// Mitsubishi GX Developer project: 11-1201_球閥後半段組立機_20140305   PLC: FX3U

PROGRAM MAIN
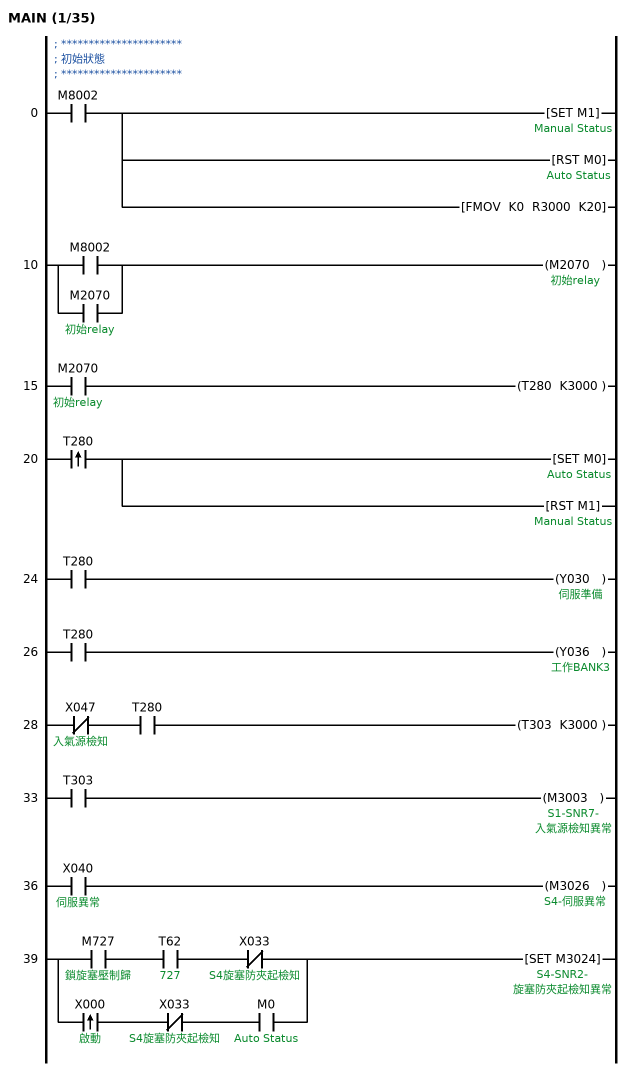
; **********************
; 初始狀態
; **********************
0     LD      M8002
      SET     M1  ; Manual Status
      RST     M0  ; Auto Status
      FMOV    K0 R3000 K20
10    LD      M8002
      OR      M2070  ; 初始relay
      OUT     M2070  ; 初始relay
15    LD      M2070  ; 初始relay
      OUT     T280 K3000
20    LDP     T280
      SET     M0  ; Auto Status
      RST     M1  ; Manual Status
24    LD      T280
      OUT     Y030  ; 伺服準備
26    LD      T280
      OUT     Y036  ; 工作BANK3
28    LDI     X047  ; 入氣源檢知
      AND     T280
      OUT     T303 K3000
33    LD      T303
      OUT     M3003  ; S1-SNR7-入氣源檢知異常
36    LD      X040  ; 伺服異常
      OUT     M3026  ; S4-伺服異常
39    LD      M727  ; 鎖旋塞壓制歸
      AND     T62  ; 727
      ANI     X033  ; S4旋塞防夾起檢知
      LDP     X000  ; 啟動
      ANI     X033  ; S4旋塞防夾起檢知
      AND     M0  ; Auto Status
      ORB
      SET     M3024  ; S4-SNR2-旋塞防夾起檢知異常
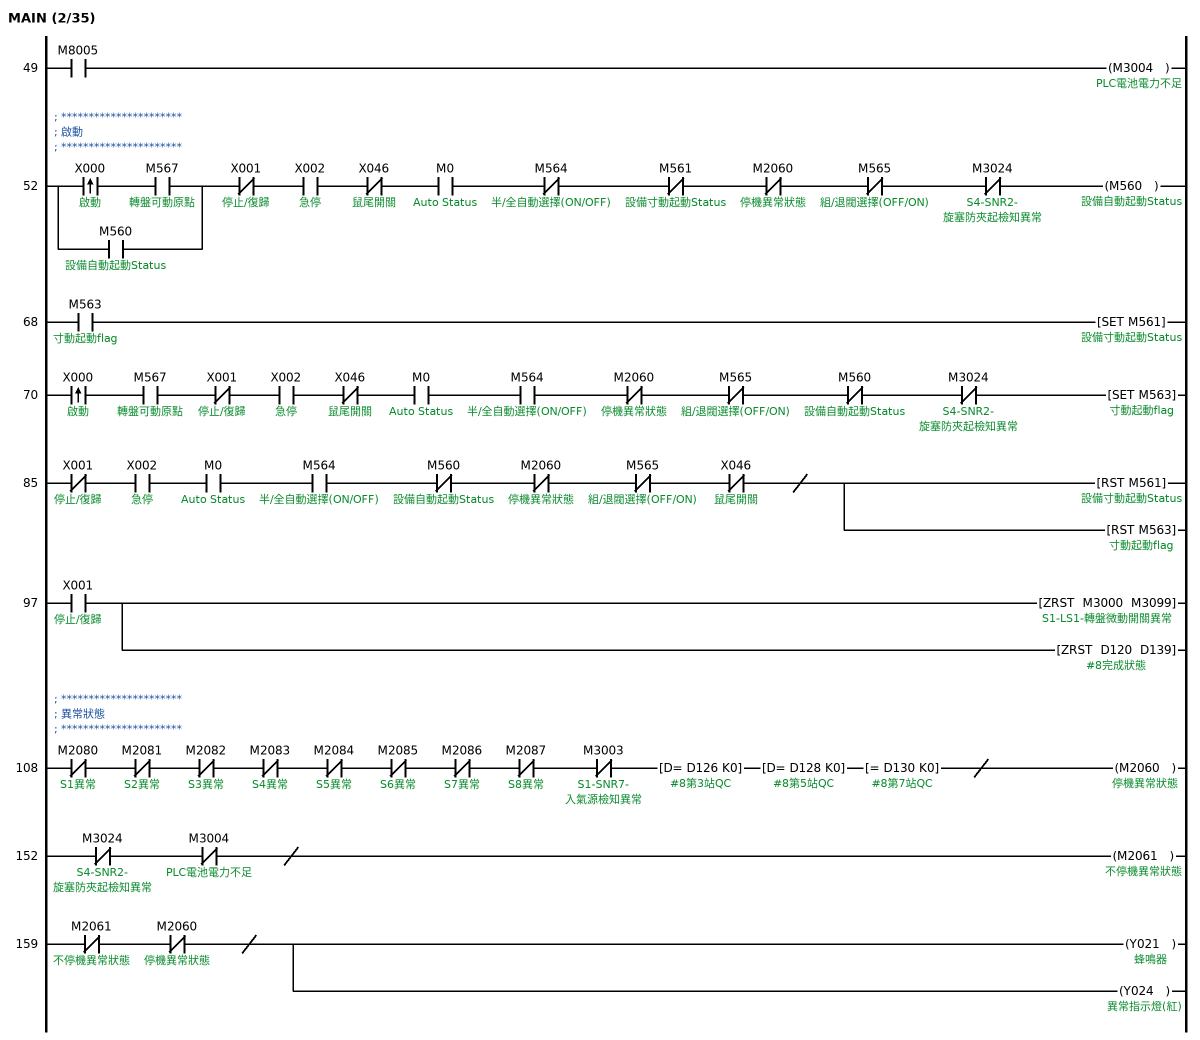
49    LD      M8005
      OUT     M3004  ; PLC電池電力不足
; **********************
; 啟動
; **********************
52    LDP     X000  ; 啟動
      AND     M567  ; 轉盤可動原點
      OR      M560  ; 設備自動起動Status
      ANI     X001  ; 停止/復歸
      AND     X002  ; 急停
      ANI     X046  ; 鼠尾開關
      AND     M0  ; Auto Status
      ANI     M564  ; 半/全自動選擇(ON/OFF)
      ANI     M561  ; 設備寸動起動Status
      ANI     M2060  ; 停機異常狀態
      ANI     M565  ; 組/退閥選擇(OFF/ON)
      ANI     M3024  ; S4-SNR2-旋塞防夾起檢知異常
      OUT     M560  ; 設備自動起動Status
68    LD      M563  ; 寸動起動flag
      SET     M561  ; 設備寸動起動Status
70    LDP     X000  ; 啟動
      AND     M567  ; 轉盤可動原點
      ANI     X001  ; 停止/復歸
      AND     X002  ; 急停
      ANI     X046  ; 鼠尾開關
      AND     M0  ; Auto Status
      AND     M564  ; 半/全自動選擇(ON/OFF)
      ANI     M2060  ; 停機異常狀態
      ANI     M565  ; 組/退閥選擇(OFF/ON)
      ANI     M560  ; 設備自動起動Status
      ANI     M3024  ; S4-SNR2-旋塞防夾起檢知異常
      SET     M563  ; 寸動起動flag
85    LDI     X001  ; 停止/復歸
      AND     X002  ; 急停
      AND     M0  ; Auto Status
      AND     M564  ; 半/全自動選擇(ON/OFF)
      ANI     M560  ; 設備自動起動Status
      ANI     M2060  ; 停機異常狀態
      ANI     M565  ; 組/退閥選擇(OFF/ON)
      ANI     X046  ; 鼠尾開關
      INV
      RST     M561  ; 設備寸動起動Status
      RST     M563  ; 寸動起動flag
97    LD      X001  ; 停止/復歸
      ZRST    M3000 M3099  ; S1-LS1-轉盤微動開關異常
      ZRST    D120 D139  ; #8完成狀態
; **********************
; 異常狀態
; **********************
108   LDI     M2080  ; S1異常
      ANI     M2081  ; S2異常
      ANI     M2082  ; S3異常
      ANI     M2083  ; S4異常
      ANI     M2084  ; S5異常
      ANI     M2085  ; S6異常
      ANI     M2086  ; S7異常
      ANI     M2087  ; S8異常
      ANI     M3003  ; S1-SNR7-入氣源檢知異常
      ANDD=   D126 K0  ; #8第3站QC
      ANDD=   D128 K0  ; #8第5站QC
      AND=    D130 K0  ; #8第7站QC
      INV
      OUT     M2060  ; 停機異常狀態
152   LDI     M3024  ; S4-SNR2-旋塞防夾起檢知異常
      ANI     M3004  ; PLC電池電力不足
      INV
      OUT     M2061  ; 不停機異常狀態
159   LDI     M2061  ; 不停機異常狀態
      ANI     M2060  ; 停機異常狀態
      INV
      OUT     Y021  ; 蜂鳴器
      OUT     Y024  ; 異常指示燈(紅)
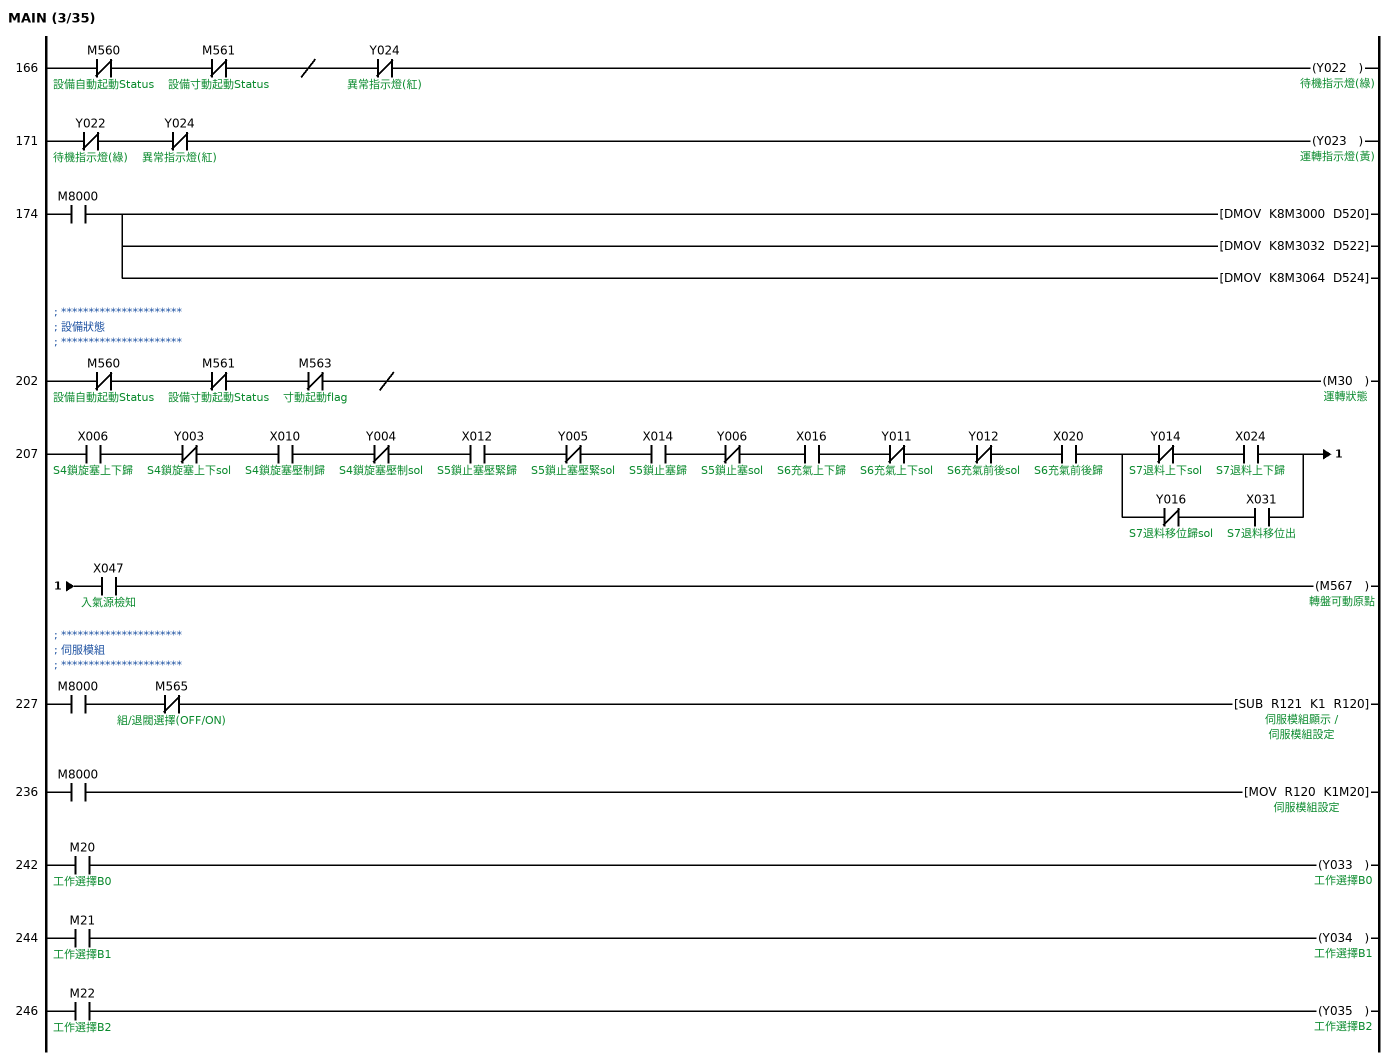
166   LDI     M560  ; 設備自動起動Status
      ANI     M561  ; 設備寸動起動Status
      INV
      ANI     Y024  ; 異常指示燈(紅)
      OUT     Y022  ; 待機指示燈(綠)
171   LDI     Y022  ; 待機指示燈(綠)
      ANI     Y024  ; 異常指示燈(紅)
      OUT     Y023  ; 運轉指示燈(黃)
174   LD      M8000
      DMOV    K8M3000 D520
      DMOV    K8M3032 D522
      DMOV    K8M3064 D524  ; S6-LS16-充氣旋轉歸異常
; **********************
; 設備狀態
; **********************
202   LDI     M560  ; 設備自動起動Status
      ANI     M561  ; 設備寸動起動Status
      ANI     M563  ; 寸動起動flag
      INV
      OUT     M30  ; 運轉狀態
207   LD      X006  ; S4鎖旋塞上下歸
      ANI     Y003  ; S4鎖旋塞上下sol
      AND     X010  ; S4鎖旋塞壓制歸
      ANI     Y004  ; S4鎖旋塞壓制sol
      AND     X012  ; S5鎖止塞壓緊歸
      ANI     Y005  ; S5鎖止塞壓緊sol
      AND     X014  ; S5鎖止塞歸
      ANI     Y006  ; S5鎖止塞sol
      AND     X016  ; S6充氣上下歸
      ANI     Y011  ; S6充氣上下sol
      ANI     Y012  ; S6充氣前後sol
      AND     X020  ; S6充氣前後歸
      LDI     Y014  ; S7退料上下sol
      AND     X024  ; S7退料上下歸
      LDI     Y016  ; S7退料移位歸sol
      AND     X031  ; S7退料移位出
      ORB
      ANB
      AND     X047  ; 入氣源檢知
      OUT     M567  ; 轉盤可動原點
; **********************
; 伺服模組
; **********************
227   LD      M8000
      ANI     M565  ; 組/退閥選擇(OFF/ON)
      SUB     R121 K1 R120  ; 伺服模組顯示 / 伺服模組設定
236   LD      M8000
      MOV     R120 K1M20  ; 工作選擇B0
242   LD      M20  ; 工作選擇B0
      OUT     Y033  ; 工作選擇B0
244   LD      M21  ; 工作選擇B1
      OUT     Y034  ; 工作選擇B1
246   LD      M22  ; 工作選擇B2
      OUT     Y035  ; 工作選擇B2
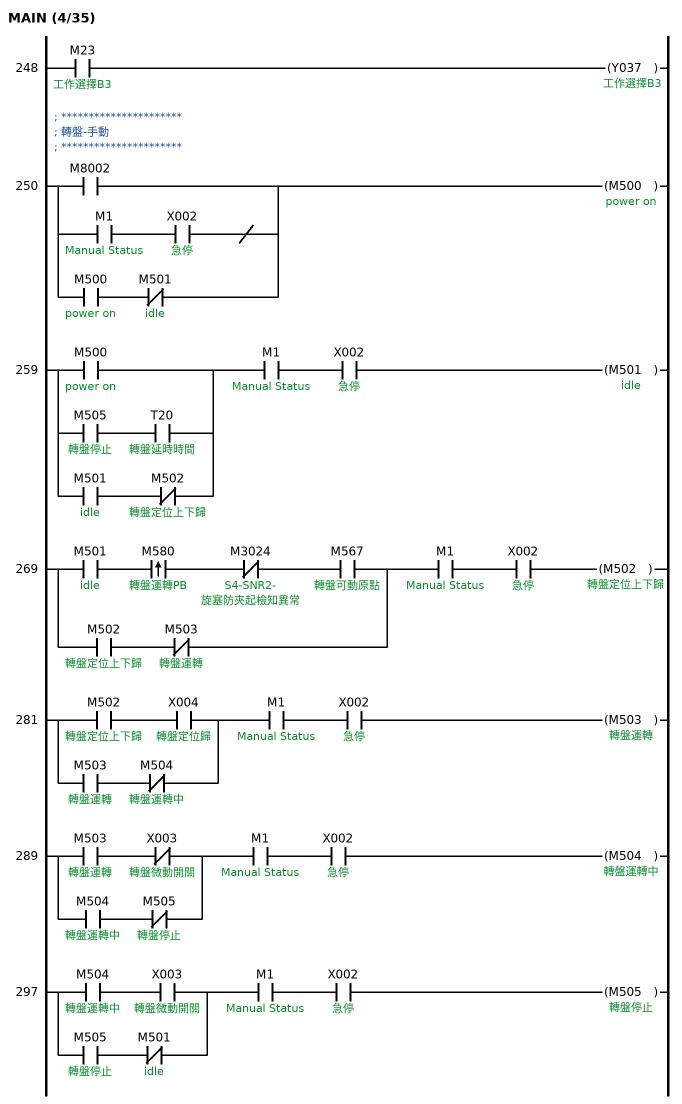
248   LD      M23  ; 工作選擇B3
      OUT     Y037  ; 工作選擇B3
; **********************
; 轉盤-手動
; **********************
250   LD      M8002
      LD      M1  ; Manual Status
      AND     X002  ; 急停
      INV
      ORB
      LD      M500  ; power on
      ANI     M501  ; idle
      ORB
      OUT     M500  ; power on
259   LD      M500  ; power on
      LD      M505  ; 轉盤停止
      AND     T20  ; 轉盤延時時間
      ORB
      LD      M501  ; idle
      ANI     M502  ; 轉盤定位上下歸
      ORB
      AND     M1  ; Manual Status
      AND     X002  ; 急停
      OUT     M501  ; idle
269   LD      M501  ; idle
      ANDP    M580  ; 轉盤運轉PB
      ANI     M3024  ; S4-SNR2-旋塞防夾起檢知異常
      AND     M567  ; 轉盤可動原點
      LD      M502  ; 轉盤定位上下歸
      ANI     M503  ; 轉盤運轉
      ORB
      AND     M1  ; Manual Status
      AND     X002  ; 急停
      OUT     M502  ; 轉盤定位上下歸
281   LD      M502  ; 轉盤定位上下歸
      AND     X004  ; 轉盤定位歸
      LD      M503  ; 轉盤運轉
      ANI     M504  ; 轉盤運轉中
      ORB
      AND     M1  ; Manual Status
      AND     X002  ; 急停
      OUT     M503  ; 轉盤運轉
289   LD      M503  ; 轉盤運轉
      ANI     X003  ; 轉盤微動開關
      LD      M504  ; 轉盤運轉中
      ANI     M505  ; 轉盤停止
      ORB
      AND     M1  ; Manual Status
      AND     X002  ; 急停
      OUT     M504  ; 轉盤運轉中
297   LD      M504  ; 轉盤運轉中
      AND     X003  ; 轉盤微動開關
      LD      M505  ; 轉盤停止
      ANI     M501  ; idle
      ORB
      AND     M1  ; Manual Status
      AND     X002  ; 急停
      OUT     M505  ; 轉盤停止
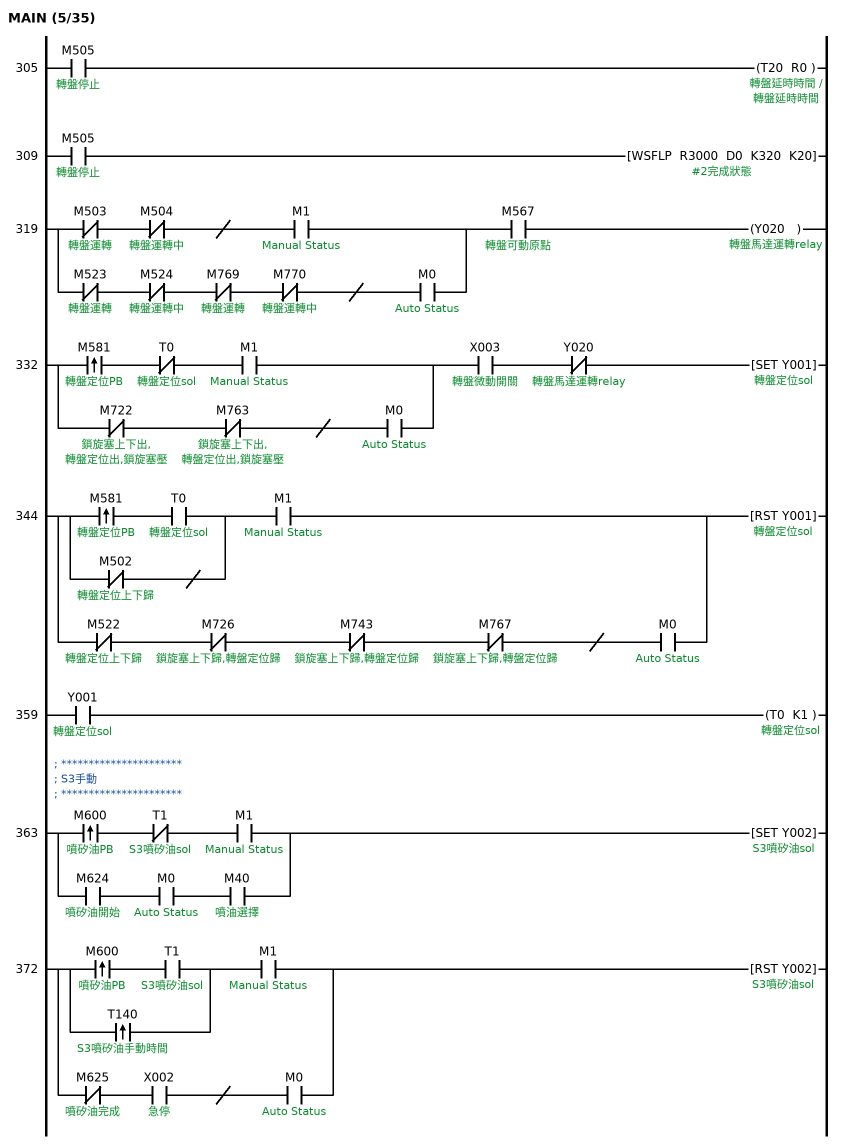
305   LD      M505  ; 轉盤停止
      OUT     T20 R0  ; 轉盤延時時間 / 轉盤延時時間
309   LD      M505  ; 轉盤停止
      WSFLP   R3000 D0 K320 K20  ; #2完成狀態
319   LDI     M503  ; 轉盤運轉
      ANI     M504  ; 轉盤運轉中
      INV
      AND     M1  ; Manual Status
      LDI     M523  ; 轉盤運轉
      ANI     M524  ; 轉盤運轉中
      ANI     M769  ; 轉盤運轉
      ANI     M770  ; 轉盤運轉中
      INV
      AND     M0  ; Auto Status
      ORB
      AND     M567  ; 轉盤可動原點
      OUT     Y020  ; 轉盤馬達運轉relay
332   LDP     M581  ; 轉盤定位PB
      ANI     T0  ; 轉盤定位sol
      AND     M1  ; Manual Status
      LDI     M722  ; 鎖旋塞上下出,轉盤定位出,鎖旋塞壓
      ANI     M763  ; 鎖旋塞上下出,轉盤定位出,鎖旋塞壓
      INV
      AND     M0  ; Auto Status
      ORB
      AND     X003  ; 轉盤微動開關
      ANI     Y020  ; 轉盤馬達運轉relay
      SET     Y001  ; 轉盤定位sol
344   LDP     M581  ; 轉盤定位PB
      AND     T0  ; 轉盤定位sol
      LDI     M502  ; 轉盤定位上下歸
      INV
      ORB
      AND     M1  ; Manual Status
      LDI     M522  ; 轉盤定位上下歸
      ANI     M726  ; 鎖旋塞上下歸,轉盤定位歸
      ANI     M743  ; 鎖旋塞上下歸,轉盤定位歸
      ANI     M767  ; 鎖旋塞上下歸,轉盤定位歸
      INV
      AND     M0  ; Auto Status
      ORB
      RST     Y001  ; 轉盤定位sol
359   LD      Y001  ; 轉盤定位sol
      OUT     T0 K1  ; 轉盤定位sol
; **********************
; S3手動
; **********************
363   LDP     M600  ; 噴矽油PB
      ANI     T1  ; S3噴矽油sol
      AND     M1  ; Manual Status
      LD      M624  ; 噴矽油開始
      AND     M0  ; Auto Status
      AND     M40  ; 噴油選擇
      ORB
      SET     Y002  ; S3噴矽油sol
372   LDP     M600  ; 噴矽油PB
      AND     T1  ; S3噴矽油sol
      ORP     T140  ; S3噴矽油手動時間
      AND     M1  ; Manual Status
      LDI     M625  ; 噴矽油完成
      AND     X002  ; 急停
      INV
      AND     M0  ; Auto Status
      ORB
      RST     Y002  ; S3噴矽油sol
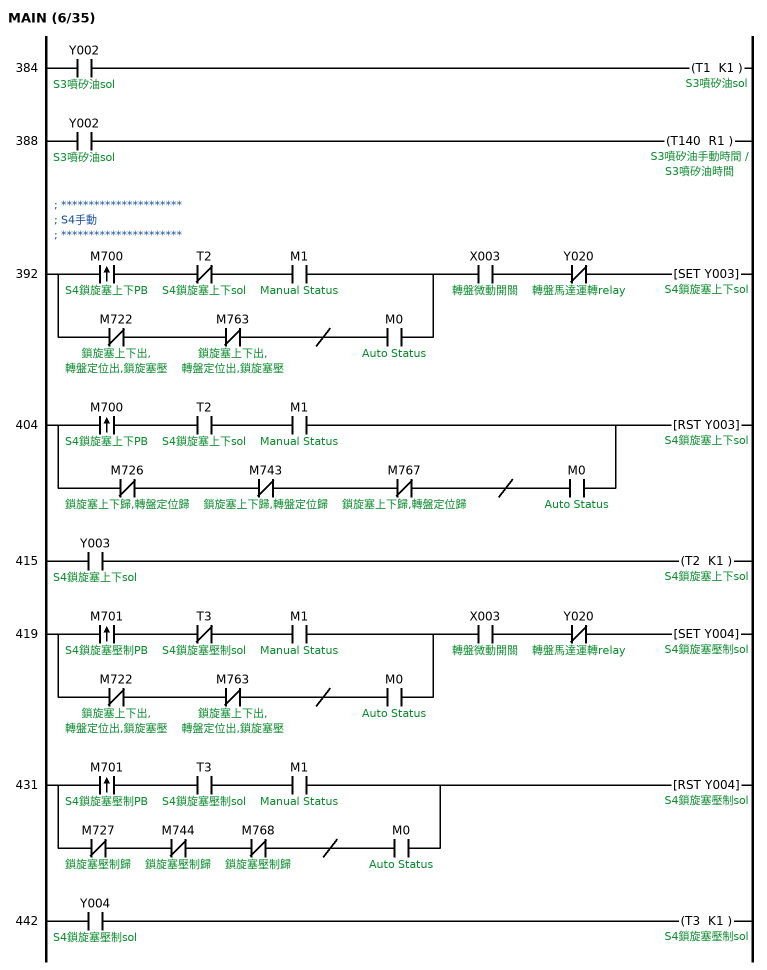
384   LD      Y002  ; S3噴矽油sol
      OUT     T1 K1  ; S3噴矽油sol
388   LD      Y002  ; S3噴矽油sol
      OUT     T140 R1  ; S3噴矽油手動時間 / S3噴矽油時間
; **********************
; S4手動
; **********************
392   LDP     M700  ; S4鎖旋塞上下PB
      ANI     T2  ; S4鎖旋塞上下sol
      AND     M1  ; Manual Status
      LDI     M722  ; 鎖旋塞上下出,轉盤定位出,鎖旋塞壓
      ANI     M763  ; 鎖旋塞上下出,轉盤定位出,鎖旋塞壓
      INV
      AND     M0  ; Auto Status
      ORB
      AND     X003  ; 轉盤微動開關
      ANI     Y020  ; 轉盤馬達運轉relay
      SET     Y003  ; S4鎖旋塞上下sol
404   LDP     M700  ; S4鎖旋塞上下PB
      AND     T2  ; S4鎖旋塞上下sol
      AND     M1  ; Manual Status
      LDI     M726  ; 鎖旋塞上下歸,轉盤定位歸
      ANI     M743  ; 鎖旋塞上下歸,轉盤定位歸
      ANI     M767  ; 鎖旋塞上下歸,轉盤定位歸
      INV
      AND     M0  ; Auto Status
      ORB
      RST     Y003  ; S4鎖旋塞上下sol
415   LD      Y003  ; S4鎖旋塞上下sol
      OUT     T2 K1  ; S4鎖旋塞上下sol
419   LDP     M701  ; S4鎖旋塞壓制PB
      ANI     T3  ; S4鎖旋塞壓制sol
      AND     M1  ; Manual Status
      LDI     M722  ; 鎖旋塞上下出,轉盤定位出,鎖旋塞壓
      ANI     M763  ; 鎖旋塞上下出,轉盤定位出,鎖旋塞壓
      INV
      AND     M0  ; Auto Status
      ORB
      AND     X003  ; 轉盤微動開關
      ANI     Y020  ; 轉盤馬達運轉relay
      SET     Y004  ; S4鎖旋塞壓制sol
431   LDP     M701  ; S4鎖旋塞壓制PB
      AND     T3  ; S4鎖旋塞壓制sol
      AND     M1  ; Manual Status
      LDI     M727  ; 鎖旋塞壓制歸
      ANI     M744  ; 鎖旋塞壓制歸
      ANI     M768  ; 鎖旋塞壓制歸
      INV
      AND     M0  ; Auto Status
      ORB
      RST     Y004  ; S4鎖旋塞壓制sol
442   LD      Y004  ; S4鎖旋塞壓制sol
      OUT     T3 K1  ; S4鎖旋塞壓制sol
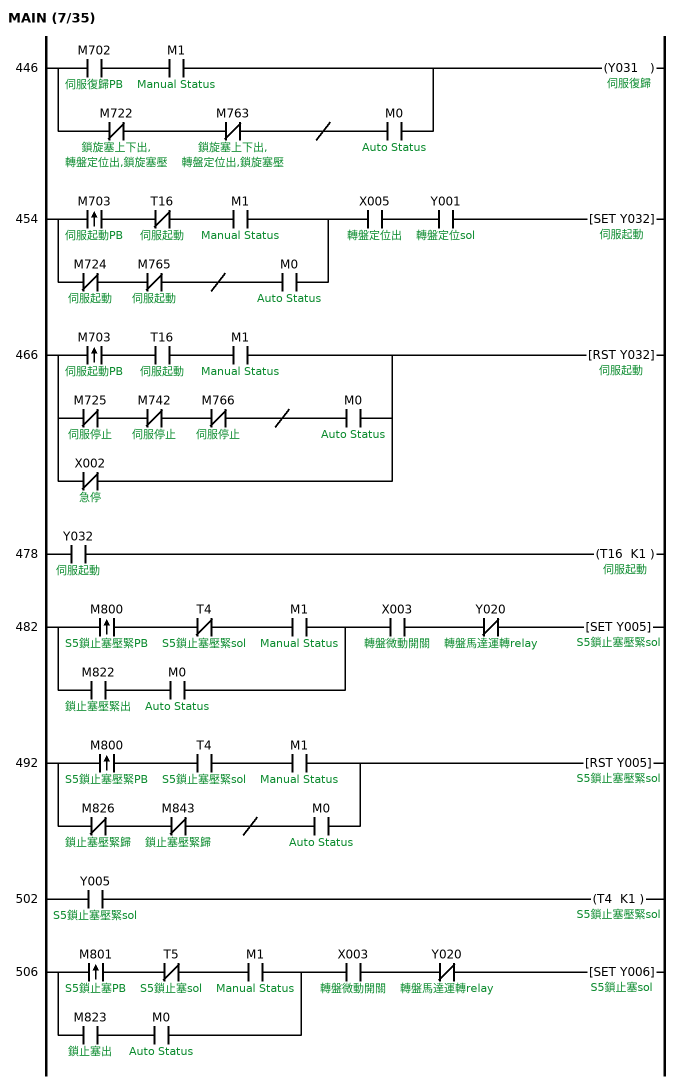
446   LD      M702  ; 伺服復歸PB
      AND     M1  ; Manual Status
      LDI     M722  ; 鎖旋塞上下出,轉盤定位出,鎖旋塞壓
      ANI     M763  ; 鎖旋塞上下出,轉盤定位出,鎖旋塞壓
      INV
      AND     M0  ; Auto Status
      ORB
      OUT     Y031  ; 伺服復歸
454   LDP     M703  ; 伺服起動PB
      ANI     T16  ; 伺服起動
      AND     M1  ; Manual Status
      LDI     M724  ; 伺服起動
      ANI     M765  ; 伺服起動
      INV
      AND     M0  ; Auto Status
      ORB
      AND     X005  ; 轉盤定位出
      AND     Y001  ; 轉盤定位sol
      SET     Y032  ; 伺服起動
466   LDP     M703  ; 伺服起動PB
      AND     T16  ; 伺服起動
      AND     M1  ; Manual Status
      LDI     M725  ; 伺服停止
      ANI     M742  ; 伺服停止
      ANI     M766  ; 伺服停止
      INV
      AND     M0  ; Auto Status
      ORB
      ORI     X002  ; 急停
      RST     Y032  ; 伺服起動
478   LD      Y032  ; 伺服起動
      OUT     T16 K1  ; 伺服起動
482   LDP     M800  ; S5鎖止塞壓緊PB
      ANI     T4  ; S5鎖止塞壓緊sol
      AND     M1  ; Manual Status
      LD      M822  ; 鎖止塞壓緊出
      AND     M0  ; Auto Status
      ORB
      AND     X003  ; 轉盤微動開關
      ANI     Y020  ; 轉盤馬達運轉relay
      SET     Y005  ; S5鎖止塞壓緊sol
492   LDP     M800  ; S5鎖止塞壓緊PB
      AND     T4  ; S5鎖止塞壓緊sol
      AND     M1  ; Manual Status
      LDI     M826  ; 鎖止塞壓緊歸
      ANI     M843  ; 鎖止塞壓緊歸
      INV
      AND     M0  ; Auto Status
      ORB
      RST     Y005  ; S5鎖止塞壓緊sol
502   LD      Y005  ; S5鎖止塞壓緊sol
      OUT     T4 K1  ; S5鎖止塞壓緊sol
506   LDP     M801  ; S5鎖止塞PB
      ANI     T5  ; S5鎖止塞sol
      AND     M1  ; Manual Status
      LD      M823  ; 鎖止塞出
      AND     M0  ; Auto Status
      ORB
      AND     X003  ; 轉盤微動開關
      ANI     Y020  ; 轉盤馬達運轉relay
      SET     Y006  ; S5鎖止塞sol
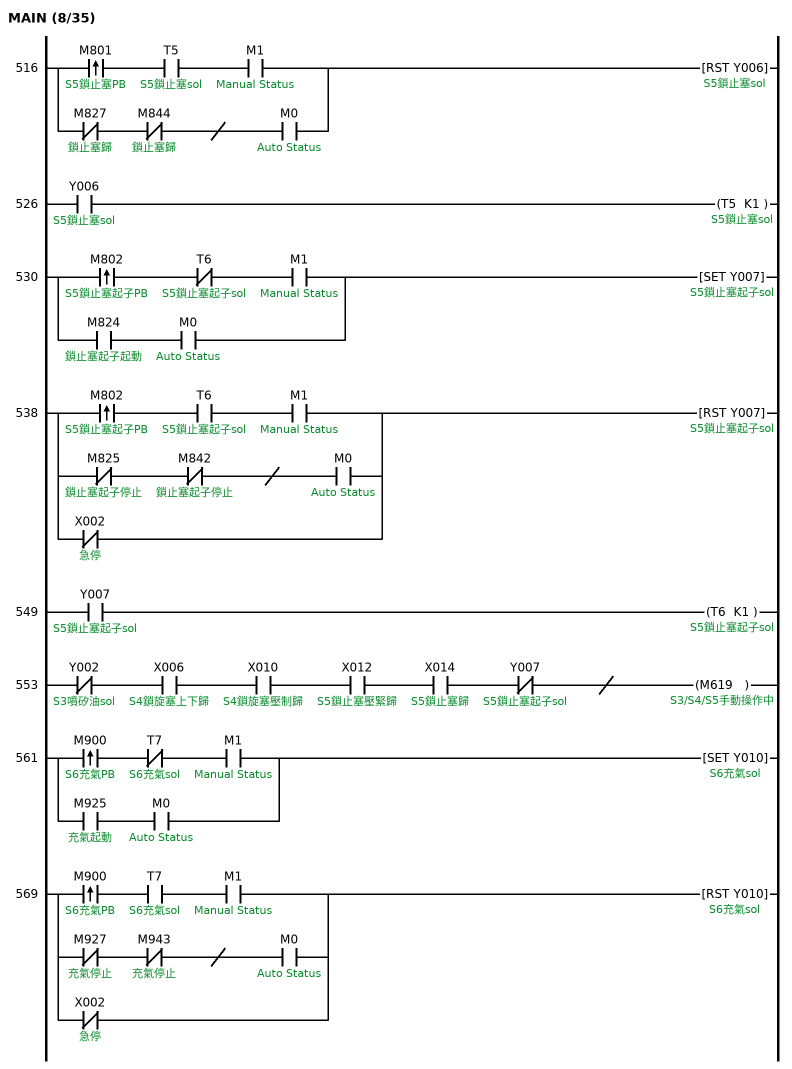
516   LDP     M801  ; S5鎖止塞PB
      AND     T5  ; S5鎖止塞sol
      AND     M1  ; Manual Status
      LDI     M827  ; 鎖止塞歸
      ANI     M844  ; 鎖止塞歸
      INV
      AND     M0  ; Auto Status
      ORB
      RST     Y006  ; S5鎖止塞sol
526   LD      Y006  ; S5鎖止塞sol
      OUT     T5 K1  ; S5鎖止塞sol
530   LDP     M802  ; S5鎖止塞起子PB
      ANI     T6  ; S5鎖止塞起子sol
      AND     M1  ; Manual Status
      LD      M824  ; 鎖止塞起子起動
      AND     M0  ; Auto Status
      ORB
      SET     Y007  ; S5鎖止塞起子sol
538   LDP     M802  ; S5鎖止塞起子PB
      AND     T6  ; S5鎖止塞起子sol
      AND     M1  ; Manual Status
      LDI     M825  ; 鎖止塞起子停止
      ANI     M842  ; 鎖止塞起子停止
      INV
      AND     M0  ; Auto Status
      ORB
      ORI     X002  ; 急停
      RST     Y007  ; S5鎖止塞起子sol
549   LD      Y007  ; S5鎖止塞起子sol
      OUT     T6 K1  ; S5鎖止塞起子sol
553   LDI     Y002  ; S3噴矽油sol
      AND     X006  ; S4鎖旋塞上下歸
      AND     X010  ; S4鎖旋塞壓制歸
      AND     X012  ; S5鎖止塞壓緊歸
      AND     X014  ; S5鎖止塞歸
      ANI     Y007  ; S5鎖止塞起子sol
      INV
      OUT     M619  ; S3/S4/S5手動操作中
561   LDP     M900  ; S6充氣PB
      ANI     T7  ; S6充氣sol
      AND     M1  ; Manual Status
      LD      M925  ; 充氣起動
      AND     M0  ; Auto Status
      ORB
      SET     Y010  ; S6充氣sol
569   LDP     M900  ; S6充氣PB
      AND     T7  ; S6充氣sol
      AND     M1  ; Manual Status
      LDI     M927  ; 充氣停止
      ANI     M943  ; 充氣停止
      INV
      AND     M0  ; Auto Status
      ORB
      ORI     X002  ; 急停
      RST     Y010  ; S6充氣sol
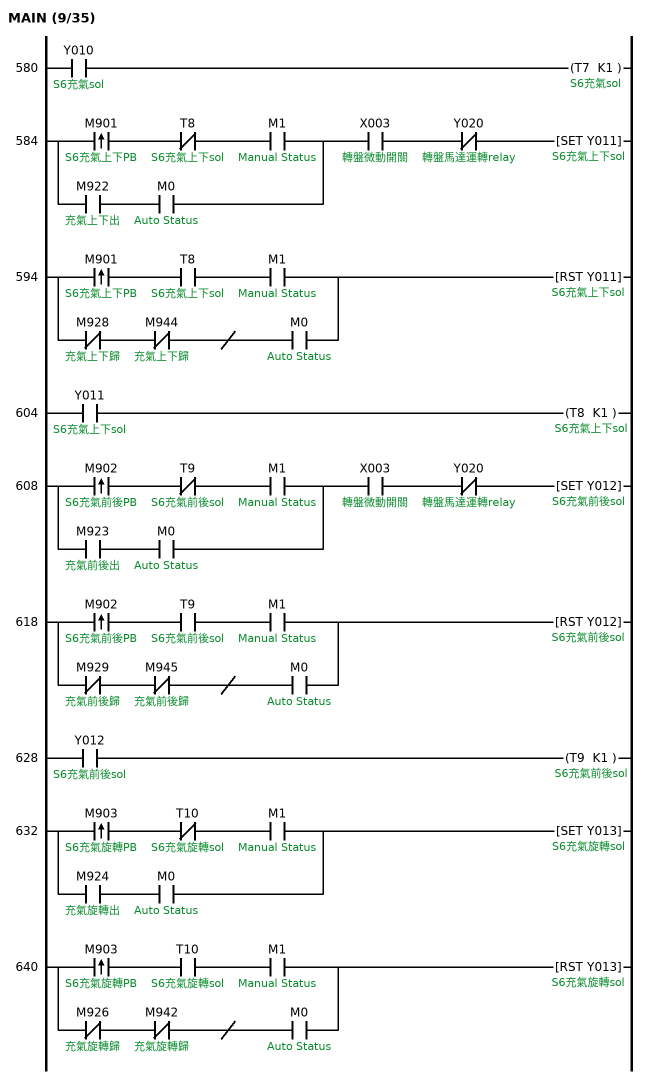
580   LD      Y010  ; S6充氣sol
      OUT     T7 K1  ; S6充氣sol
584   LDP     M901  ; S6充氣上下PB
      ANI     T8  ; S6充氣上下sol
      AND     M1  ; Manual Status
      LD      M922  ; 充氣上下出
      AND     M0  ; Auto Status
      ORB
      AND     X003  ; 轉盤微動開關
      ANI     Y020  ; 轉盤馬達運轉relay
      SET     Y011  ; S6充氣上下sol
594   LDP     M901  ; S6充氣上下PB
      AND     T8  ; S6充氣上下sol
      AND     M1  ; Manual Status
      LDI     M928  ; 充氣上下歸
      ANI     M944  ; 充氣上下歸
      INV
      AND     M0  ; Auto Status
      ORB
      RST     Y011  ; S6充氣上下sol
604   LD      Y011  ; S6充氣上下sol
      OUT     T8 K1  ; S6充氣上下sol
608   LDP     M902  ; S6充氣前後PB
      ANI     T9  ; S6充氣前後sol
      AND     M1  ; Manual Status
      LD      M923  ; 充氣前後出
      AND     M0  ; Auto Status
      ORB
      AND     X003  ; 轉盤微動開關
      ANI     Y020  ; 轉盤馬達運轉relay
      SET     Y012  ; S6充氣前後sol
618   LDP     M902  ; S6充氣前後PB
      AND     T9  ; S6充氣前後sol
      AND     M1  ; Manual Status
      LDI     M929  ; 充氣前後歸
      ANI     M945  ; 充氣前後歸
      INV
      AND     M0  ; Auto Status
      ORB
      RST     Y012  ; S6充氣前後sol
628   LD      Y012  ; S6充氣前後sol
      OUT     T9 K1  ; S6充氣前後sol
632   LDP     M903  ; S6充氣旋轉PB
      ANI     T10  ; S6充氣旋轉sol
      AND     M1  ; Manual Status
      LD      M924  ; 充氣旋轉出
      AND     M0  ; Auto Status
      ORB
      SET     Y013  ; S6充氣旋轉sol
640   LDP     M903  ; S6充氣旋轉PB
      AND     T10  ; S6充氣旋轉sol
      AND     M1  ; Manual Status
      LDI     M926  ; 充氣旋轉歸
      ANI     M942  ; 充氣旋轉歸
      INV
      AND     M0  ; Auto Status
      ORB
      RST     Y013  ; S6充氣旋轉sol
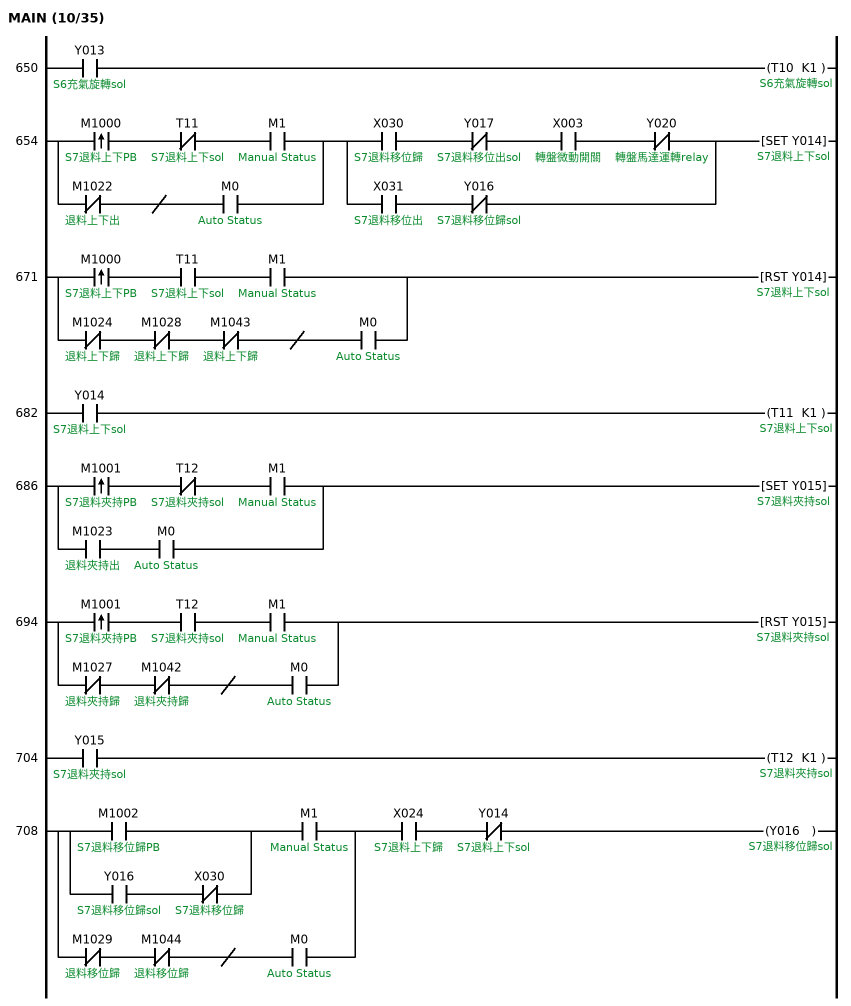
650   LD      Y013  ; S6充氣旋轉sol
      OUT     T10 K1  ; S6充氣旋轉sol
654   LDP     M1000  ; S7退料上下PB
      ANI     T11  ; S7退料上下sol
      AND     M1  ; Manual Status
      LDI     M1022  ; 退料上下出
      INV
      AND     M0  ; Auto Status
      ORB
      LD      X030  ; S7退料移位歸
      ANI     Y017  ; S7退料移位出sol
      AND     X003  ; 轉盤微動開關
      ANI     Y020  ; 轉盤馬達運轉relay
      LD      X031  ; S7退料移位出
      ANI     Y016  ; S7退料移位歸sol
      ORB
      ANB
      SET     Y014  ; S7退料上下sol
671   LDP     M1000  ; S7退料上下PB
      AND     T11  ; S7退料上下sol
      AND     M1  ; Manual Status
      LDI     M1024  ; 退料上下歸
      ANI     M1028  ; 退料上下歸
      ANI     M1043  ; 退料上下歸
      INV
      AND     M0  ; Auto Status
      ORB
      RST     Y014  ; S7退料上下sol
682   LD      Y014  ; S7退料上下sol
      OUT     T11 K1  ; S7退料上下sol
686   LDP     M1001  ; S7退料夾持PB
      ANI     T12  ; S7退料夾持sol
      AND     M1  ; Manual Status
      LD      M1023  ; 退料夾持出
      AND     M0  ; Auto Status
      ORB
      SET     Y015  ; S7退料夾持sol
694   LDP     M1001  ; S7退料夾持PB
      AND     T12  ; S7退料夾持sol
      AND     M1  ; Manual Status
      LDI     M1027  ; 退料夾持歸
      ANI     M1042  ; 退料夾持歸
      INV
      AND     M0  ; Auto Status
      ORB
      RST     Y015  ; S7退料夾持sol
704   LD      Y015  ; S7退料夾持sol
      OUT     T12 K1  ; S7退料夾持sol
708   LD      M1002  ; S7退料移位歸PB
      LD      Y016  ; S7退料移位歸sol
      ANI     X030  ; S7退料移位歸
      ORB
      AND     M1  ; Manual Status
      LDI     M1029  ; 退料移位歸
      ANI     M1044  ; 退料移位歸
      INV
      AND     M0  ; Auto Status
      ORB
      AND     X024  ; S7退料上下歸
      ANI     Y014  ; S7退料上下sol
      OUT     Y016  ; S7退料移位歸sol
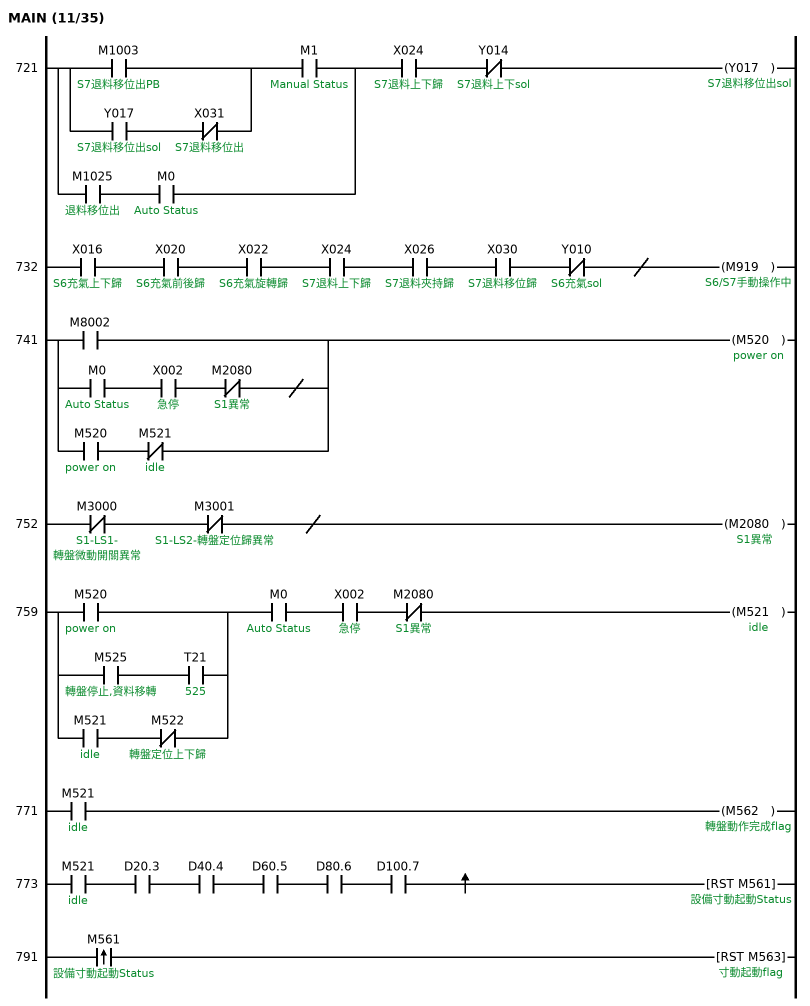
721   LD      M1003  ; S7退料移位出PB
      LD      Y017  ; S7退料移位出sol
      ANI     X031  ; S7退料移位出
      ORB
      AND     M1  ; Manual Status
      LD      M1025  ; 退料移位出
      AND     M0  ; Auto Status
      ORB
      AND     X024  ; S7退料上下歸
      ANI     Y014  ; S7退料上下sol
      OUT     Y017  ; S7退料移位出sol
732   LD      X016  ; S6充氣上下歸
      AND     X020  ; S6充氣前後歸
      AND     X022  ; S6充氣旋轉歸
      AND     X024  ; S7退料上下歸
      AND     X026  ; S7退料夾持歸
      AND     X030  ; S7退料移位歸
      ANI     Y010  ; S6充氣sol
      INV
      OUT     M919  ; S6/S7手動操作中
741   LD      M8002
      LD      M0  ; Auto Status
      AND     X002  ; 急停
      ANI     M2080  ; S1異常
      INV
      ORB
      LD      M520  ; power on
      ANI     M521  ; idle
      ORB
      OUT     M520  ; power on
752   LDI     M3000  ; S1-LS1-轉盤微動開關異常
      ANI     M3001  ; S1-LS2-轉盤定位歸異常
      INV
      OUT     M2080  ; S1異常
759   LD      M520  ; power on
      LD      M525  ; 轉盤停止,資料移轉
      AND     T21  ; 525
      ORB
      LD      M521  ; idle
      ANI     M522  ; 轉盤定位上下歸
      ORB
      AND     M0  ; Auto Status
      AND     X002  ; 急停
      ANI     M2080  ; S1異常
      OUT     M521  ; idle
771   LD      M521  ; idle
      OUT     M562  ; 轉盤動作完成flag
773   LD      M521  ; idle
      AND     D20.3
      AND     D40.4
      AND     D60.5
      AND     D80.6
      AND     D100.7
      MEP
      RST     M561  ; 設備寸動起動Status
791   LDP     M561  ; 設備寸動起動Status
      RST     M563  ; 寸動起動flag
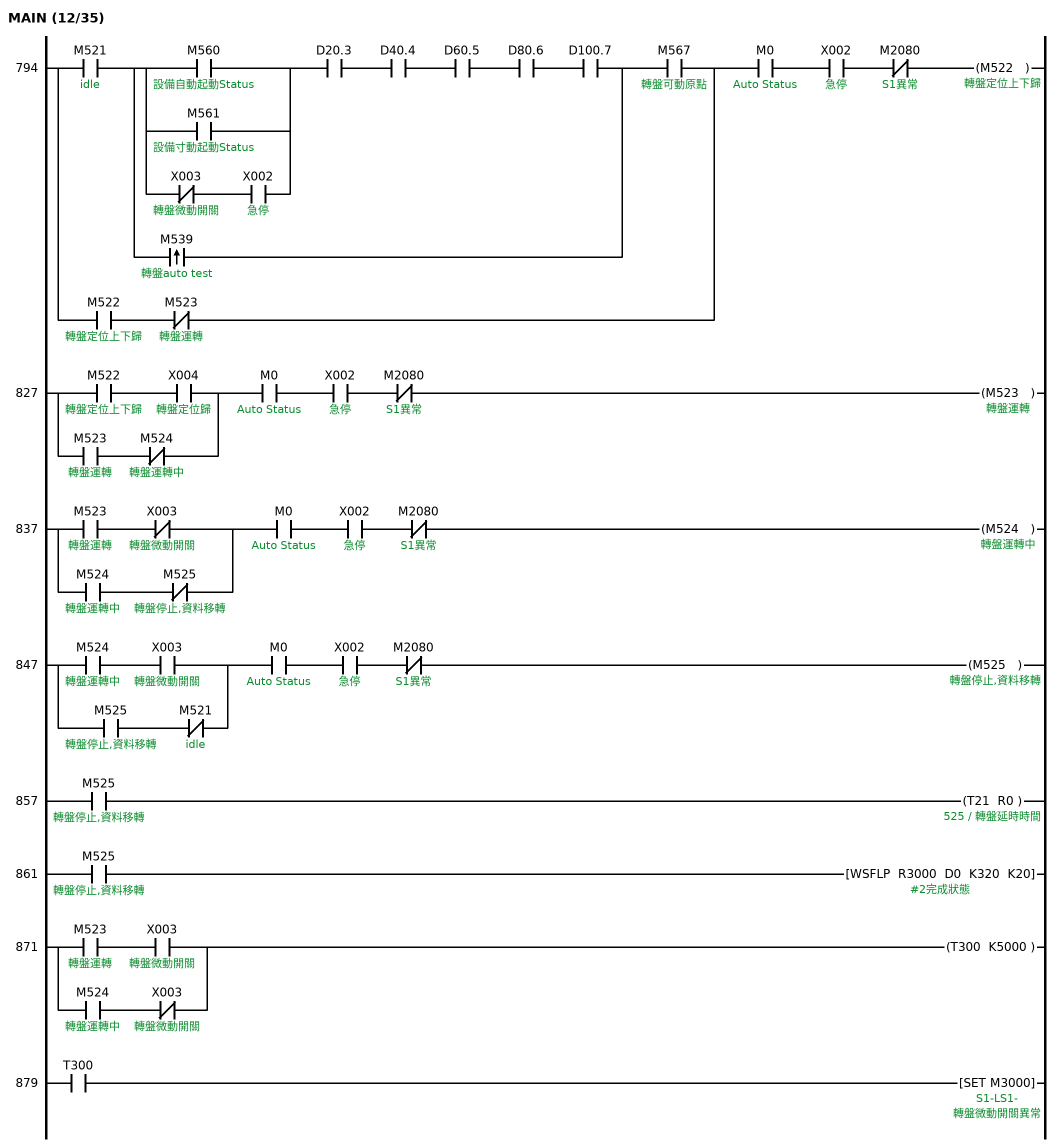
794   LD      M521  ; idle
      LD      M560  ; 設備自動起動Status
      OR      M561  ; 設備寸動起動Status
      LDI     X003  ; 轉盤微動開關
      AND     X002  ; 急停
      ORB
      AND     D20.3
      AND     D40.4
      AND     D60.5
      AND     D80.6
      AND     D100.7
      ORP     M539  ; 轉盤auto test
      ANB
      AND     M567  ; 轉盤可動原點
      LD      M522  ; 轉盤定位上下歸
      ANI     M523  ; 轉盤運轉
      ORB
      AND     M0  ; Auto Status
      AND     X002  ; 急停
      ANI     M2080  ; S1異常
      OUT     M522  ; 轉盤定位上下歸
827   LD      M522  ; 轉盤定位上下歸
      AND     X004  ; 轉盤定位歸
      LD      M523  ; 轉盤運轉
      ANI     M524  ; 轉盤運轉中
      ORB
      AND     M0  ; Auto Status
      AND     X002  ; 急停
      ANI     M2080  ; S1異常
      OUT     M523  ; 轉盤運轉
837   LD      M523  ; 轉盤運轉
      ANI     X003  ; 轉盤微動開關
      LD      M524  ; 轉盤運轉中
      ANI     M525  ; 轉盤停止,資料移轉
      ORB
      AND     M0  ; Auto Status
      AND     X002  ; 急停
      ANI     M2080  ; S1異常
      OUT     M524  ; 轉盤運轉中
847   LD      M524  ; 轉盤運轉中
      AND     X003  ; 轉盤微動開關
      LD      M525  ; 轉盤停止,資料移轉
      ANI     M521  ; idle
      ORB
      AND     M0  ; Auto Status
      AND     X002  ; 急停
      ANI     M2080  ; S1異常
      OUT     M525  ; 轉盤停止,資料移轉
857   LD      M525  ; 轉盤停止,資料移轉
      OUT     T21 R0  ; 525 / 轉盤延時時間
861   LD      M525  ; 轉盤停止,資料移轉
      WSFLP   R3000 D0 K320 K20
871   LD      M523  ; 轉盤運轉
      AND     X003  ; 轉盤微動開關
      LD      M524  ; 轉盤運轉中
      ANI     X003  ; 轉盤微動開關
      ORB
      OUT     T300 K5000
879   LD      T300
      SET     M3000  ; S1-LS1-轉盤微動開關異常
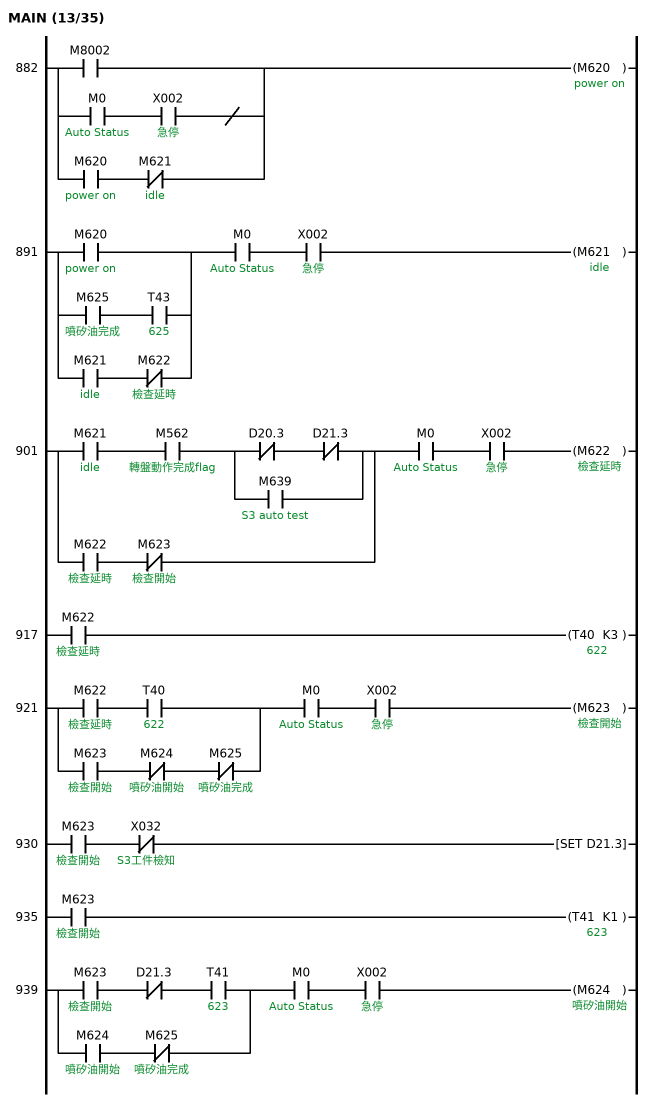
882   LD      M8002
      LD      M0  ; Auto Status
      AND     X002  ; 急停
      INV
      ORB
      LD      M620  ; power on
      ANI     M621  ; idle
      ORB
      OUT     M620  ; power on
891   LD      M620  ; power on
      LD      M625  ; 噴矽油完成
      AND     T43  ; 625
      ORB
      LD      M621  ; idle
      ANI     M622  ; 檢查延時
      ORB
      AND     M0  ; Auto Status
      AND     X002  ; 急停
      OUT     M621  ; idle
901   LD      M621  ; idle
      AND     M562  ; 轉盤動作完成flag
      LDI     D20.3
      ANI     D21.3
      OR      M639  ; S3 auto test
      ANB
      LD      M622  ; 檢查延時
      ANI     M623  ; 檢查開始
      ORB
      AND     M0  ; Auto Status
      AND     X002  ; 急停
      OUT     M622  ; 檢查延時
917   LD      M622  ; 檢查延時
      OUT     T40 K3  ; 622
921   LD      M622  ; 檢查延時
      AND     T40  ; 622
      LD      M623  ; 檢查開始
      ANI     M624  ; 噴矽油開始
      ANI     M625  ; 噴矽油完成
      ORB
      AND     M0  ; Auto Status
      AND     X002  ; 急停
      OUT     M623  ; 檢查開始
930   LD      M623  ; 檢查開始
      ANI     X032  ; S3工件檢知
      SET     D21.3
935   LD      M623  ; 檢查開始
      OUT     T41 K1  ; 623
939   LD      M623  ; 檢查開始
      ANI     D21.3
      AND     T41  ; 623
      LD      M624  ; 噴矽油開始
      ANI     M625  ; 噴矽油完成
      ORB
      AND     M0  ; Auto Status
      AND     X002  ; 急停
      OUT     M624  ; 噴矽油開始
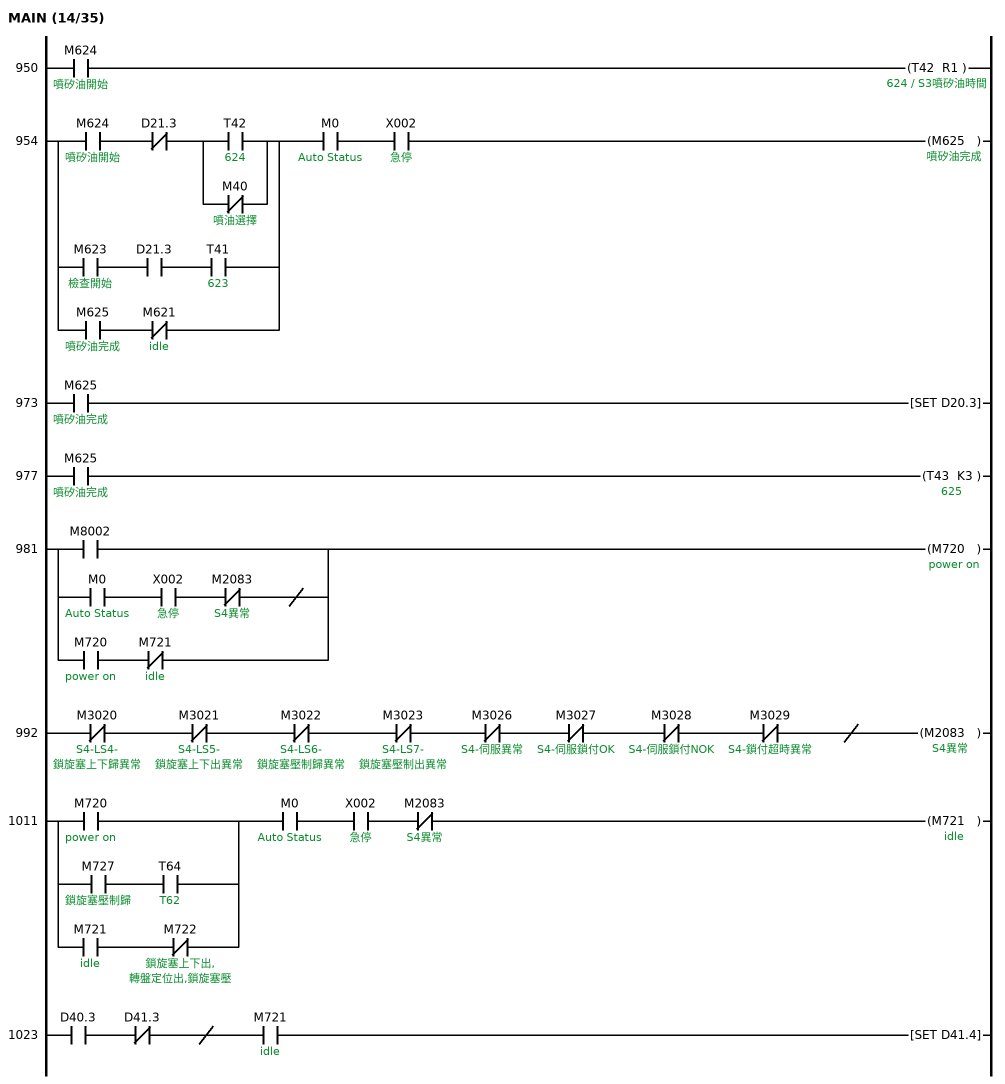
950   LD      M624  ; 噴矽油開始
      OUT     T42 R1  ; 624 / S3噴矽油時間
954   LD      M624  ; 噴矽油開始
      ANI     D21.3
      LD      T42  ; 624
      ORI     M40  ; 噴油選擇
      ANB
      LD      M623  ; 檢查開始
      AND     D21.3
      AND     T41  ; 623
      ORB
      LD      M625  ; 噴矽油完成
      ANI     M621  ; idle
      ORB
      AND     M0  ; Auto Status
      AND     X002  ; 急停
      OUT     M625  ; 噴矽油完成
973   LD      M625  ; 噴矽油完成
      SET     D20.3
977   LD      M625  ; 噴矽油完成
      OUT     T43 K3  ; 625
981   LD      M8002
      LD      M0  ; Auto Status
      AND     X002  ; 急停
      ANI     M2083  ; S4異常
      INV
      ORB
      LD      M720  ; power on
      ANI     M721  ; idle
      ORB
      OUT     M720  ; power on
992   LDI     M3020  ; S4-LS4-鎖旋塞上下歸異常
      ANI     M3021  ; S4-LS5-鎖旋塞上下出異常
      ANI     M3022  ; S4-LS6-鎖旋塞壓制歸異常
      ANI     M3023  ; S4-LS7-鎖旋塞壓制出異常
      ANI     M3026  ; S4-伺服異常
      ANI     M3027  ; S4-伺服鎖付OK
      ANI     M3028  ; S4-伺服鎖付NOK
      ANI     M3029  ; S4-鎖付超時異常
      INV
      OUT     M2083  ; S4異常
1011  LD      M720  ; power on
      LD      M727  ; 鎖旋塞壓制歸
      AND     T64  ; T62
      ORB
      LD      M721  ; idle
      ANI     M722  ; 鎖旋塞上下出,轉盤定位出,鎖旋塞壓
      ORB
      AND     M0  ; Auto Status
      AND     X002  ; 急停
      ANI     M2083  ; S4異常
      OUT     M721  ; idle
1023  LD      D40.3
      ANI     D41.3
      INV
      AND     M721  ; idle
      SET     D41.4
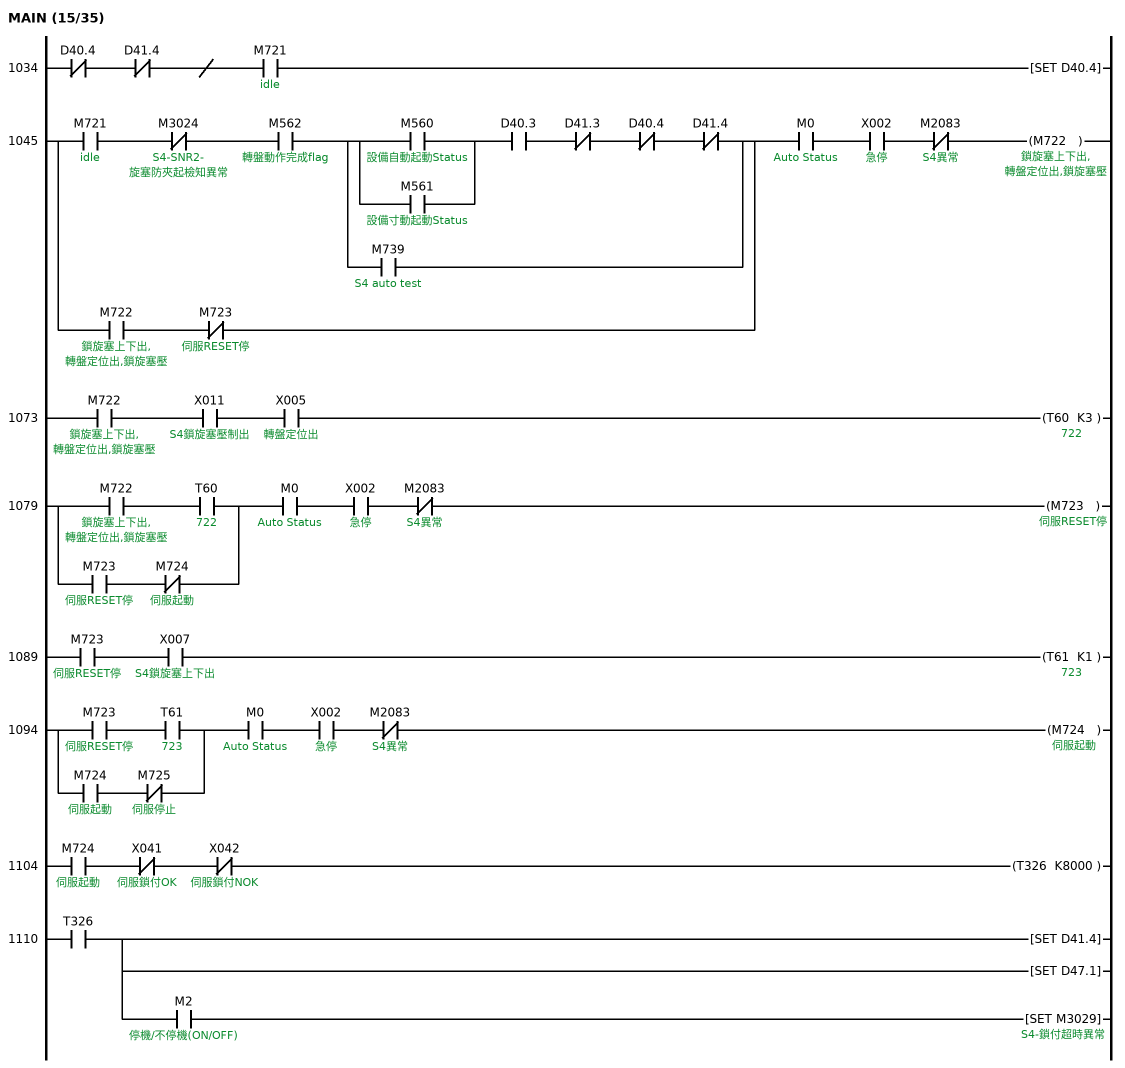
1034  LDI     D40.4
      ANI     D41.4
      INV
      AND     M721  ; idle
      SET     D40.4
1045  LD      M721  ; idle
      ANI     M3024  ; S4-SNR2-旋塞防夾起檢知異常
      AND     M562  ; 轉盤動作完成flag
      LD      M560  ; 設備自動起動Status
      OR      M561  ; 設備寸動起動Status
      AND     D40.3
      ANI     D41.3
      ANI     D40.4
      ANI     D41.4
      OR      M739  ; S4 auto test
      ANB
      LD      M722  ; 鎖旋塞上下出,轉盤定位出,鎖旋塞壓
      ANI     M723  ; 伺服RESET停
      ORB
      AND     M0  ; Auto Status
      AND     X002  ; 急停
      ANI     M2083  ; S4異常
      OUT     M722  ; 鎖旋塞上下出,轉盤定位出,鎖旋塞壓
1073  LD      M722  ; 鎖旋塞上下出,轉盤定位出,鎖旋塞壓
      AND     X011  ; S4鎖旋塞壓制出
      AND     X005  ; 轉盤定位出
      OUT     T60 K3  ; 722
1079  LD      M722  ; 鎖旋塞上下出,轉盤定位出,鎖旋塞壓
      AND     T60  ; 722
      LD      M723  ; 伺服RESET停
      ANI     M724  ; 伺服起動
      ORB
      AND     M0  ; Auto Status
      AND     X002  ; 急停
      ANI     M2083  ; S4異常
      OUT     M723  ; 伺服RESET停
1089  LD      M723  ; 伺服RESET停
      AND     X007  ; S4鎖旋塞上下出
      OUT     T61 K1  ; 723
1094  LD      M723  ; 伺服RESET停
      AND     T61  ; 723
      LD      M724  ; 伺服起動
      ANI     M725  ; 伺服停止
      ORB
      AND     M0  ; Auto Status
      AND     X002  ; 急停
      ANI     M2083  ; S4異常
      OUT     M724  ; 伺服起動
1104  LD      M724  ; 伺服起動
      ANI     X041  ; 伺服鎖付OK
      ANI     X042  ; 伺服鎖付NOK
      OUT     T326 K8000
1110  LD      T326
      SET     D41.4
      SET     D47.1
      AND     M2  ; 停機/不停機(ON/OFF)
      SET     M3029  ; S4-鎖付超時異常
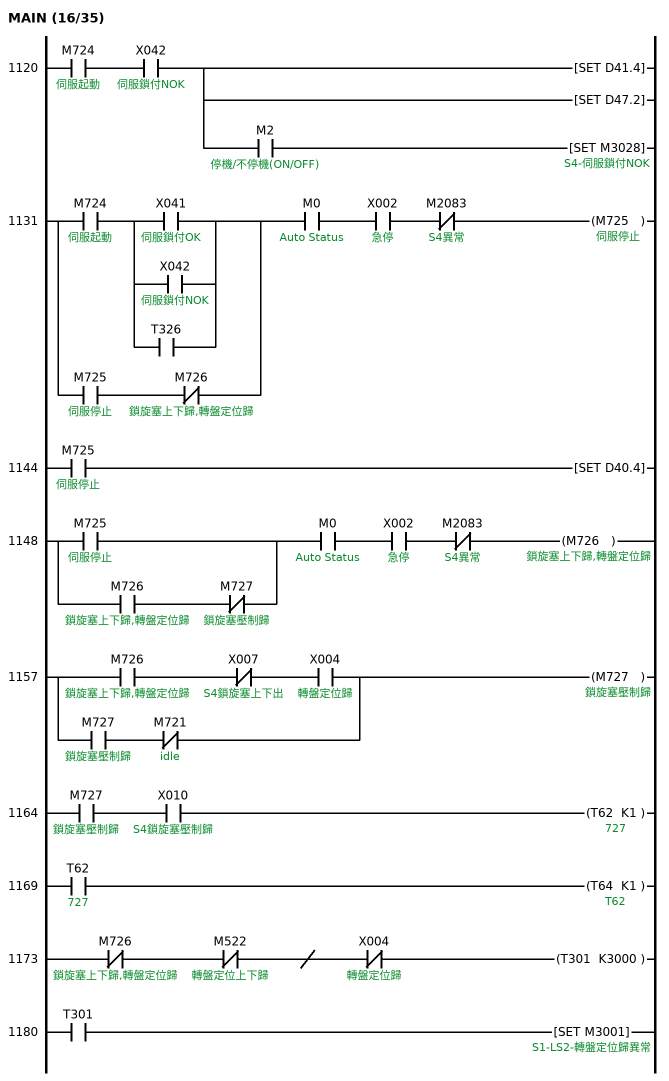
1120  LD      M724  ; 伺服起動
      AND     X042  ; 伺服鎖付NOK
      SET     D41.4
      SET     D47.2
      AND     M2  ; 停機/不停機(ON/OFF)
      SET     M3028  ; S4-伺服鎖付NOK
1131  LD      M724  ; 伺服起動
      LD      X041  ; 伺服鎖付OK
      OR      X042  ; 伺服鎖付NOK
      OR      T326
      ANB
      LD      M725  ; 伺服停止
      ANI     M726  ; 鎖旋塞上下歸,轉盤定位歸
      ORB
      AND     M0  ; Auto Status
      AND     X002  ; 急停
      ANI     M2083  ; S4異常
      OUT     M725  ; 伺服停止
1144  LD      M725  ; 伺服停止
      SET     D40.4
1148  LD      M725  ; 伺服停止
      LD      M726  ; 鎖旋塞上下歸,轉盤定位歸
      ANI     M727  ; 鎖旋塞壓制歸
      ORB
      AND     M0  ; Auto Status
      AND     X002  ; 急停
      ANI     M2083  ; S4異常
      OUT     M726  ; 鎖旋塞上下歸,轉盤定位歸
1157  LD      M726  ; 鎖旋塞上下歸,轉盤定位歸
      ANI     X007  ; S4鎖旋塞上下出
      AND     X004  ; 轉盤定位歸
      LD      M727  ; 鎖旋塞壓制歸
      ANI     M721  ; idle
      ORB
      OUT     M727  ; 鎖旋塞壓制歸
1164  LD      M727  ; 鎖旋塞壓制歸
      AND     X010  ; S4鎖旋塞壓制歸
      OUT     T62 K1  ; 727
1169  LD      T62  ; 727
      OUT     T64 K1  ; T62
1173  LDI     M726  ; 鎖旋塞上下歸,轉盤定位歸
      ANI     M522  ; 轉盤定位上下歸
      INV
      ANI     X004  ; 轉盤定位歸
      OUT     T301 K3000
1180  LD      T301
      SET     M3001  ; S1-LS2-轉盤定位歸異常
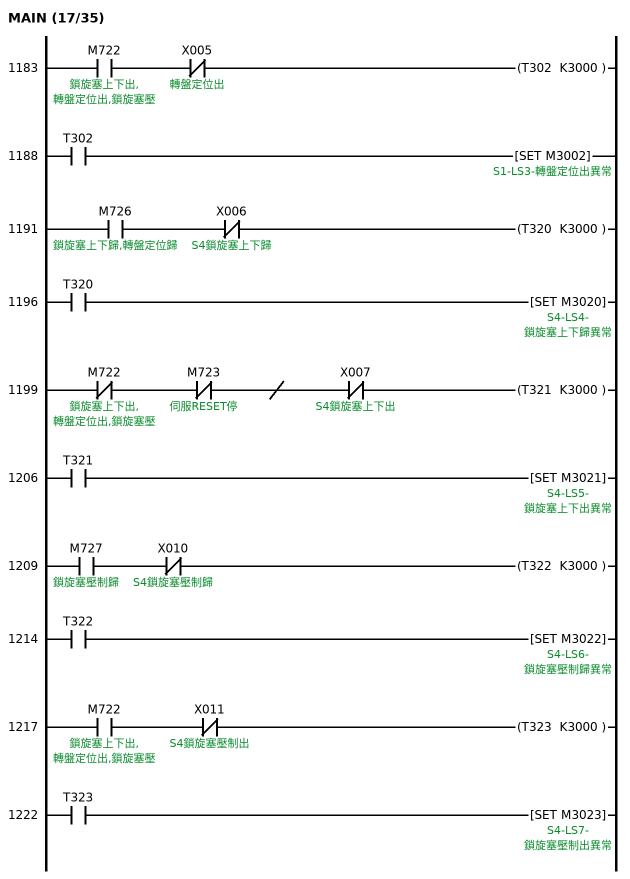
1183  LD      M722  ; 鎖旋塞上下出,轉盤定位出,鎖旋塞壓
      ANI     X005  ; 轉盤定位出
      OUT     T302 K3000
1188  LD      T302
      SET     M3002  ; S1-LS3-轉盤定位出異常
1191  LD      M726  ; 鎖旋塞上下歸,轉盤定位歸
      ANI     X006  ; S4鎖旋塞上下歸
      OUT     T320 K3000
1196  LD      T320
      SET     M3020  ; S4-LS4-鎖旋塞上下歸異常
1199  LDI     M722  ; 鎖旋塞上下出,轉盤定位出,鎖旋塞壓
      ANI     M723  ; 伺服RESET停
      INV
      ANI     X007  ; S4鎖旋塞上下出
      OUT     T321 K3000
1206  LD      T321
      SET     M3021  ; S4-LS5-鎖旋塞上下出異常
1209  LD      M727  ; 鎖旋塞壓制歸
      ANI     X010  ; S4鎖旋塞壓制歸
      OUT     T322 K3000
1214  LD      T322
      SET     M3022  ; S4-LS6-鎖旋塞壓制歸異常
1217  LD      M722  ; 鎖旋塞上下出,轉盤定位出,鎖旋塞壓
      ANI     X011  ; S4鎖旋塞壓制出
      OUT     T323 K3000
1222  LD      T323
      SET     M3023  ; S4-LS7-鎖旋塞壓制出異常
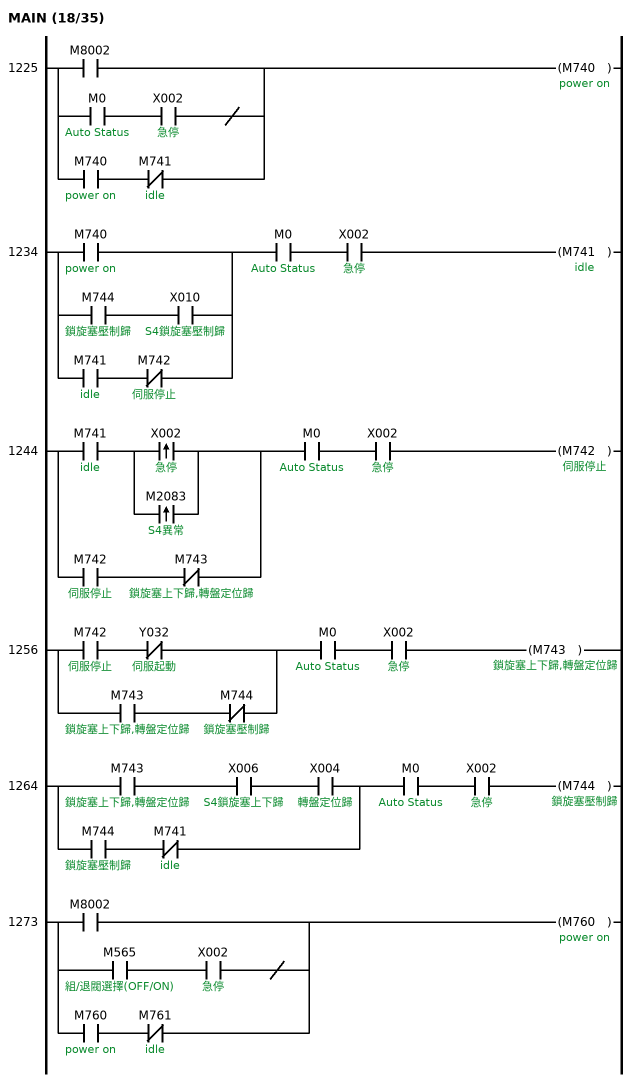
1225  LD      M8002
      LD      M0  ; Auto Status
      AND     X002  ; 急停
      INV
      ORB
      LD      M740  ; power on
      ANI     M741  ; idle
      ORB
      OUT     M740  ; power on
1234  LD      M740  ; power on
      LD      M744  ; 鎖旋塞壓制歸
      AND     X010  ; S4鎖旋塞壓制歸
      ORB
      LD      M741  ; idle
      ANI     M742  ; 伺服停止
      ORB
      AND     M0  ; Auto Status
      AND     X002  ; 急停
      OUT     M741  ; idle
1244  LD      M741  ; idle
      LDP     X002  ; 急停
      ORP     M2083  ; S4異常
      ANB
      LD      M742  ; 伺服停止
      ANI     M743  ; 鎖旋塞上下歸,轉盤定位歸
      ORB
      AND     M0  ; Auto Status
      AND     X002  ; 急停
      OUT     M742  ; 伺服停止
1256  LD      M742  ; 伺服停止
      ANI     Y032  ; 伺服起動
      LD      M743  ; 鎖旋塞上下歸,轉盤定位歸
      ANI     M744  ; 鎖旋塞壓制歸
      ORB
      AND     M0  ; Auto Status
      AND     X002  ; 急停
      OUT     M743  ; 鎖旋塞上下歸,轉盤定位歸
1264  LD      M743  ; 鎖旋塞上下歸,轉盤定位歸
      AND     X006  ; S4鎖旋塞上下歸
      AND     X004  ; 轉盤定位歸
      LD      M744  ; 鎖旋塞壓制歸
      ANI     M741  ; idle
      ORB
      AND     M0  ; Auto Status
      AND     X002  ; 急停
      OUT     M744  ; 鎖旋塞壓制歸
1273  LD      M8002
      LD      M565  ; 組/退閥選擇(OFF/ON)
      AND     X002  ; 急停
      INV
      ORB
      LD      M760  ; power on
      ANI     M761  ; idle
      ORB
      OUT     M760  ; power on
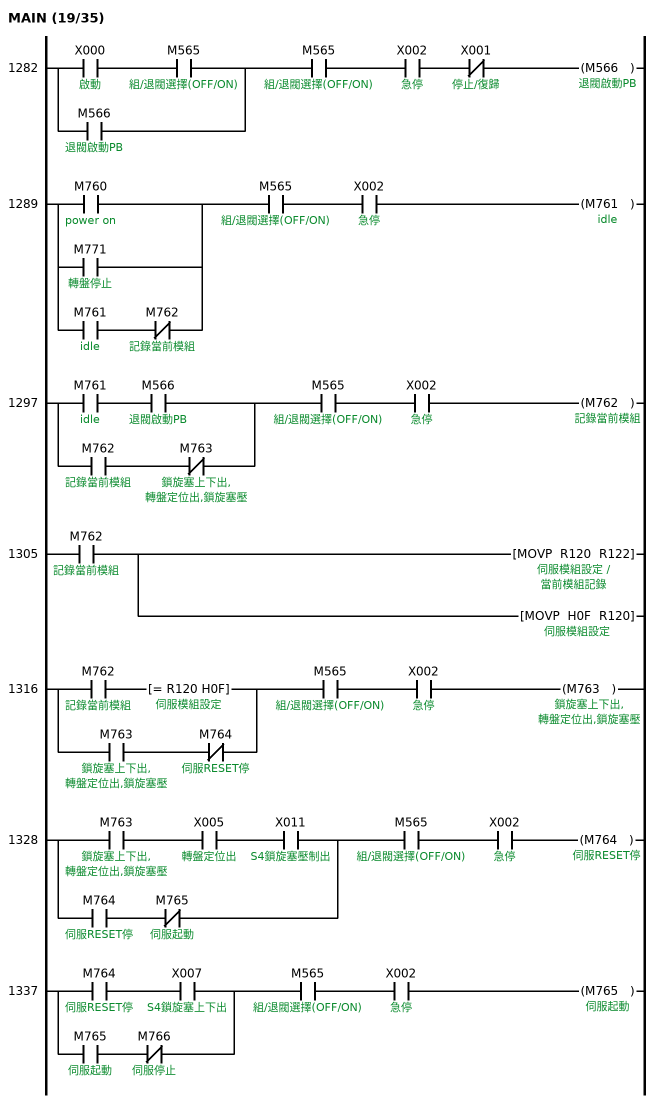
1282  LD      X000  ; 啟動
      AND     M565  ; 組/退閥選擇(OFF/ON)
      OR      M566  ; 退閥啟動PB
      AND     M565  ; 組/退閥選擇(OFF/ON)
      AND     X002  ; 急停
      ANI     X001  ; 停止/復歸
      OUT     M566  ; 退閥啟動PB
1289  LD      M760  ; power on
      OR      M771  ; 轉盤停止
      LD      M761  ; idle
      ANI     M762  ; 記錄當前模組
      ORB
      AND     M565  ; 組/退閥選擇(OFF/ON)
      AND     X002  ; 急停
      OUT     M761  ; idle
1297  LD      M761  ; idle
      AND     M566  ; 退閥啟動PB
      LD      M762  ; 記錄當前模組
      ANI     M763  ; 鎖旋塞上下出,轉盤定位出,鎖旋塞壓
      ORB
      AND     M565  ; 組/退閥選擇(OFF/ON)
      AND     X002  ; 急停
      OUT     M762  ; 記錄當前模組
1305  LD      M762  ; 記錄當前模組
      MOVP    R120 R122  ; 當前模組記錄
      MOVP    H0F R120
1316  LD      M762  ; 記錄當前模組
      AND=    R120 H0F  ; 伺服模組設定
      LD      M763  ; 鎖旋塞上下出,轉盤定位出,鎖旋塞壓
      ANI     M764  ; 伺服RESET停
      ORB
      AND     M565  ; 組/退閥選擇(OFF/ON)
      AND     X002  ; 急停
      OUT     M763  ; 鎖旋塞上下出,轉盤定位出,鎖旋塞壓
1328  LD      M763  ; 鎖旋塞上下出,轉盤定位出,鎖旋塞壓
      AND     X005  ; 轉盤定位出
      AND     X011  ; S4鎖旋塞壓制出
      LD      M764  ; 伺服RESET停
      ANI     M765  ; 伺服起動
      ORB
      AND     M565  ; 組/退閥選擇(OFF/ON)
      AND     X002  ; 急停
      OUT     M764  ; 伺服RESET停
1337  LD      M764  ; 伺服RESET停
      AND     X007  ; S4鎖旋塞上下出
      LD      M765  ; 伺服起動
      ANI     M766  ; 伺服停止
      ORB
      AND     M565  ; 組/退閥選擇(OFF/ON)
      AND     X002  ; 急停
      OUT     M765  ; 伺服起動
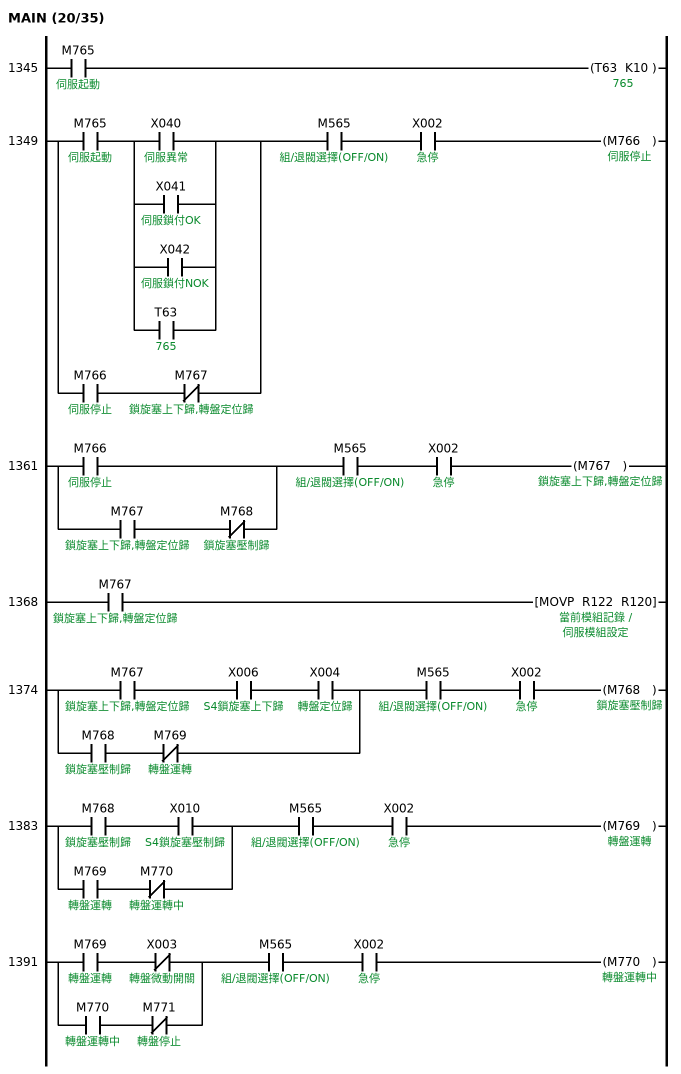
1345  LD      M765  ; 伺服起動
      OUT     T63 K10  ; 765
1349  LD      M765  ; 伺服起動
      LD      X040  ; 伺服異常
      OR      X041  ; 伺服鎖付OK
      OR      X042  ; 伺服鎖付NOK
      OR      T63  ; 765
      ANB
      LD      M766  ; 伺服停止
      ANI     M767  ; 鎖旋塞上下歸,轉盤定位歸
      ORB
      AND     M565  ; 組/退閥選擇(OFF/ON)
      AND     X002  ; 急停
      OUT     M766  ; 伺服停止
1361  LD      M766  ; 伺服停止
      LD      M767  ; 鎖旋塞上下歸,轉盤定位歸
      ANI     M768  ; 鎖旋塞壓制歸
      ORB
      AND     M565  ; 組/退閥選擇(OFF/ON)
      AND     X002  ; 急停
      OUT     M767  ; 鎖旋塞上下歸,轉盤定位歸
1368  LD      M767  ; 鎖旋塞上下歸,轉盤定位歸
      MOVP    R122 R120
1374  LD      M767  ; 鎖旋塞上下歸,轉盤定位歸
      AND     X006  ; S4鎖旋塞上下歸
      AND     X004  ; 轉盤定位歸
      LD      M768  ; 鎖旋塞壓制歸
      ANI     M769  ; 轉盤運轉
      ORB
      AND     M565  ; 組/退閥選擇(OFF/ON)
      AND     X002  ; 急停
      OUT     M768  ; 鎖旋塞壓制歸
1383  LD      M768  ; 鎖旋塞壓制歸
      AND     X010  ; S4鎖旋塞壓制歸
      LD      M769  ; 轉盤運轉
      ANI     M770  ; 轉盤運轉中
      ORB
      AND     M565  ; 組/退閥選擇(OFF/ON)
      AND     X002  ; 急停
      OUT     M769  ; 轉盤運轉
1391  LD      M769  ; 轉盤運轉
      ANI     X003  ; 轉盤微動開關
      LD      M770  ; 轉盤運轉中
      ANI     M771  ; 轉盤停止
      ORB
      AND     M565  ; 組/退閥選擇(OFF/ON)
      AND     X002  ; 急停
      OUT     M770  ; 轉盤運轉中
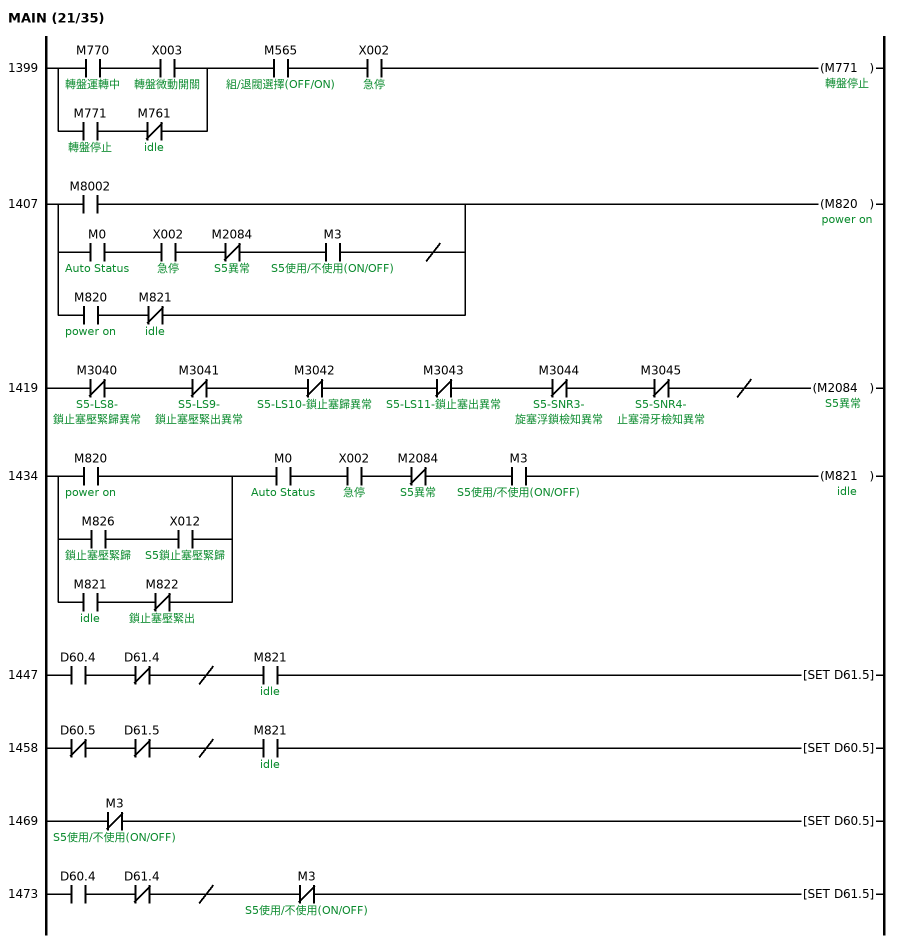
1399  LD      M770  ; 轉盤運轉中
      AND     X003  ; 轉盤微動開關
      LD      M771  ; 轉盤停止
      ANI     M761  ; idle
      ORB
      AND     M565  ; 組/退閥選擇(OFF/ON)
      AND     X002  ; 急停
      OUT     M771  ; 轉盤停止
1407  LD      M8002
      LD      M0  ; Auto Status
      AND     X002  ; 急停
      ANI     M2084  ; S5異常
      AND     M3  ; S5使用/不使用(ON/OFF)
      INV
      ORB
      LD      M820  ; power on
      ANI     M821  ; idle
      ORB
      OUT     M820  ; power on
1419  LDI     M3040  ; S5-LS8-鎖止塞壓緊歸異常
      ANI     M3041  ; S5-LS9-鎖止塞壓緊出異常
      ANI     M3042  ; S5-LS10-鎖止塞歸異常
      ANI     M3043  ; S5-LS11-鎖止塞出異常
      ANI     M3044  ; S5-SNR3-旋塞浮鎖檢知異常
      ANI     M3045  ; S5-SNR4-止塞滑牙檢知異常
      INV
      OUT     M2084  ; S5異常
1434  LD      M820  ; power on
      LD      M826  ; 鎖止塞壓緊歸
      AND     X012  ; S5鎖止塞壓緊歸
      ORB
      LD      M821  ; idle
      ANI     M822  ; 鎖止塞壓緊出
      ORB
      AND     M0  ; Auto Status
      AND     X002  ; 急停
      ANI     M2084  ; S5異常
      AND     M3  ; S5使用/不使用(ON/OFF)
      OUT     M821  ; idle
1447  LD      D60.4
      ANI     D61.4
      INV
      AND     M821  ; idle
      SET     D61.5
1458  LDI     D60.5
      ANI     D61.5
      INV
      AND     M821  ; idle
      SET     D60.5
1469  LDI     M3  ; S5使用/不使用(ON/OFF)
      SET     D60.5
1473  LD      D60.4
      ANI     D61.4
      INV
      ANI     M3  ; S5使用/不使用(ON/OFF)
      SET     D61.5
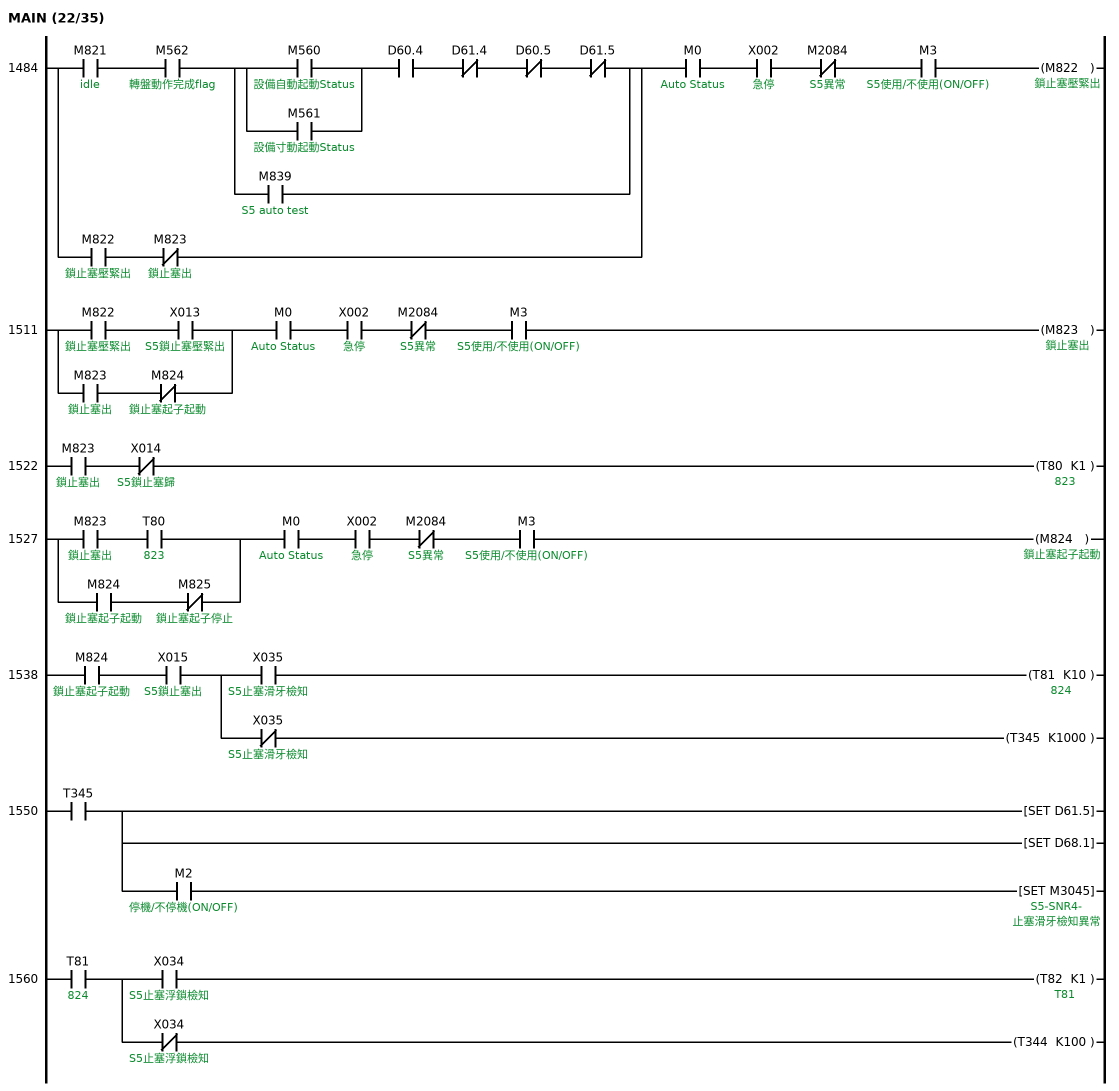
1484  LD      M821  ; idle
      AND     M562  ; 轉盤動作完成flag
      LD      M560  ; 設備自動起動Status
      OR      M561  ; 設備寸動起動Status
      AND     D60.4
      ANI     D61.4
      ANI     D60.5
      ANI     D61.5
      OR      M839  ; S5 auto test
      ANB
      LD      M822  ; 鎖止塞壓緊出
      ANI     M823  ; 鎖止塞出
      ORB
      AND     M0  ; Auto Status
      AND     X002  ; 急停
      ANI     M2084  ; S5異常
      AND     M3  ; S5使用/不使用(ON/OFF)
      OUT     M822  ; 鎖止塞壓緊出
1511  LD      M822  ; 鎖止塞壓緊出
      AND     X013  ; S5鎖止塞壓緊出
      LD      M823  ; 鎖止塞出
      ANI     M824  ; 鎖止塞起子起動
      ORB
      AND     M0  ; Auto Status
      AND     X002  ; 急停
      ANI     M2084  ; S5異常
      AND     M3  ; S5使用/不使用(ON/OFF)
      OUT     M823  ; 鎖止塞出
1522  LD      M823  ; 鎖止塞出
      ANI     X014  ; S5鎖止塞歸
      OUT     T80 K1  ; 823
1527  LD      M823  ; 鎖止塞出
      AND     T80  ; 823
      LD      M824  ; 鎖止塞起子起動
      ANI     M825  ; 鎖止塞起子停止
      ORB
      AND     M0  ; Auto Status
      AND     X002  ; 急停
      ANI     M2084  ; S5異常
      AND     M3  ; S5使用/不使用(ON/OFF)
      OUT     M824  ; 鎖止塞起子起動
1538  LD      M824  ; 鎖止塞起子起動
      AND     X015  ; S5鎖止塞出
      MPS
      AND     X035  ; S5止塞滑牙檢知
      OUT     T81 K10  ; 824
      MPP
      ANI     X035  ; S5止塞滑牙檢知
      OUT     T345 K1000
1550  LD      T345
      SET     D61.5
      SET     D68.1
      AND     M2  ; 停機/不停機(ON/OFF)
      SET     M3045  ; S5-SNR4-止塞滑牙檢知異常
1560  LD      T81  ; 824
      MPS
      AND     X034  ; S5止塞浮鎖檢知
      OUT     T82 K1  ; T81
      MPP
      ANI     X034  ; S5止塞浮鎖檢知
      OUT     T344 K100
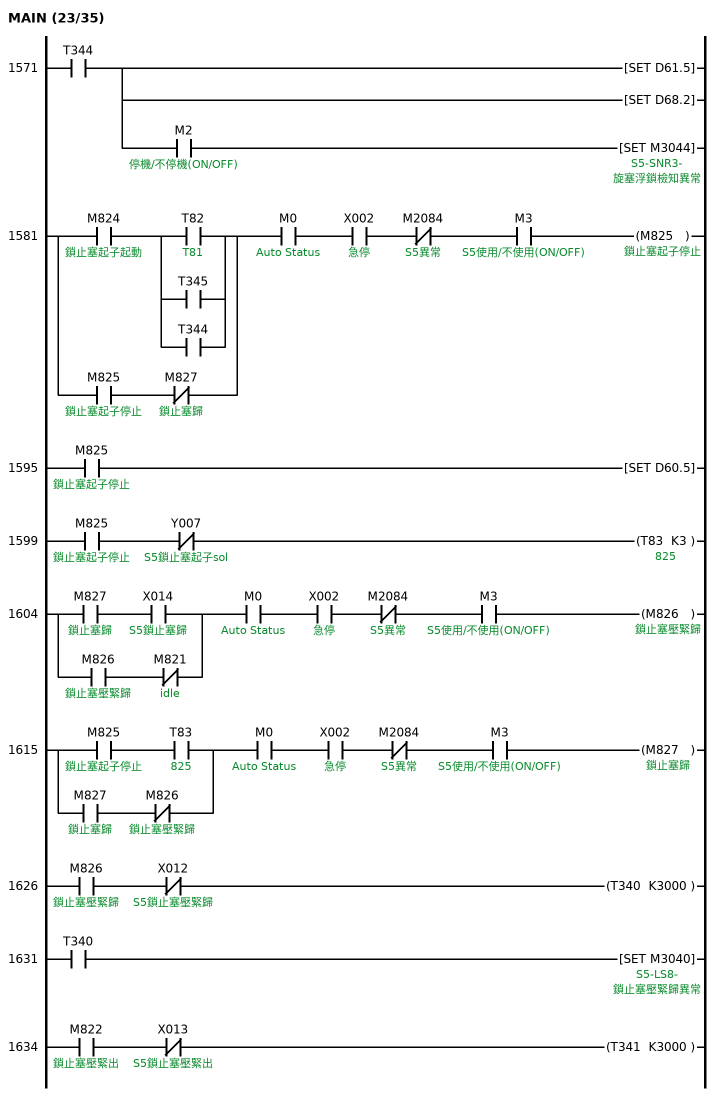
1571  LD      T344
      SET     D61.5
      SET     D68.2
      AND     M2  ; 停機/不停機(ON/OFF)
      SET     M3044  ; S5-SNR3-旋塞浮鎖檢知異常
1581  LD      M824  ; 鎖止塞起子起動
      LD      T82  ; T81
      OR      T345
      OR      T344
      ANB
      LD      M825  ; 鎖止塞起子停止
      ANI     M827  ; 鎖止塞歸
      ORB
      AND     M0  ; Auto Status
      AND     X002  ; 急停
      ANI     M2084  ; S5異常
      AND     M3  ; S5使用/不使用(ON/OFF)
      OUT     M825  ; 鎖止塞起子停止
1595  LD      M825  ; 鎖止塞起子停止
      SET     D60.5
1599  LD      M825  ; 鎖止塞起子停止
      ANI     Y007  ; S5鎖止塞起子sol
      OUT     T83 K3  ; 825
1604  LD      M827  ; 鎖止塞歸
      AND     X014  ; S5鎖止塞歸
      LD      M826  ; 鎖止塞壓緊歸
      ANI     M821  ; idle
      ORB
      AND     M0  ; Auto Status
      AND     X002  ; 急停
      ANI     M2084  ; S5異常
      AND     M3  ; S5使用/不使用(ON/OFF)
      OUT     M826  ; 鎖止塞壓緊歸
1615  LD      M825  ; 鎖止塞起子停止
      AND     T83  ; 825
      LD      M827  ; 鎖止塞歸
      ANI     M826  ; 鎖止塞壓緊歸
      ORB
      AND     M0  ; Auto Status
      AND     X002  ; 急停
      ANI     M2084  ; S5異常
      AND     M3  ; S5使用/不使用(ON/OFF)
      OUT     M827  ; 鎖止塞歸
1626  LD      M826  ; 鎖止塞壓緊歸
      ANI     X012  ; S5鎖止塞壓緊歸
      OUT     T340 K3000
1631  LD      T340
      SET     M3040  ; S5-LS8-鎖止塞壓緊歸異常
1634  LD      M822  ; 鎖止塞壓緊出
      ANI     X013  ; S5鎖止塞壓緊出
      OUT     T341 K3000
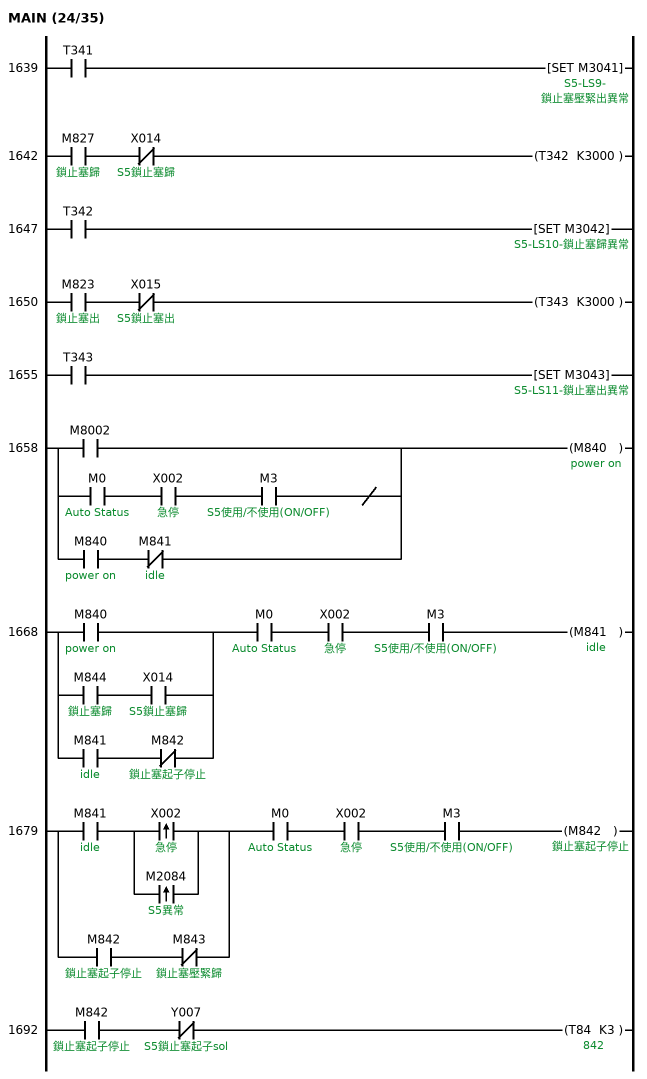
1639  LD      T341
      SET     M3041  ; S5-LS9-鎖止塞壓緊出異常
1642  LD      M827  ; 鎖止塞歸
      ANI     X014  ; S5鎖止塞歸
      OUT     T342 K3000
1647  LD      T342
      SET     M3042  ; S5-LS10-鎖止塞歸異常
1650  LD      M823  ; 鎖止塞出
      ANI     X015  ; S5鎖止塞出
      OUT     T343 K3000
1655  LD      T343
      SET     M3043  ; S5-LS11-鎖止塞出異常
1658  LD      M8002
      LD      M0  ; Auto Status
      AND     X002  ; 急停
      AND     M3  ; S5使用/不使用(ON/OFF)
      INV
      ORB
      LD      M840  ; power on
      ANI     M841  ; idle
      ORB
      OUT     M840  ; power on
1668  LD      M840  ; power on
      LD      M844  ; 鎖止塞歸
      AND     X014  ; S5鎖止塞歸
      ORB
      LD      M841  ; idle
      ANI     M842  ; 鎖止塞起子停止
      ORB
      AND     M0  ; Auto Status
      AND     X002  ; 急停
      AND     M3  ; S5使用/不使用(ON/OFF)
      OUT     M841  ; idle
1679  LD      M841  ; idle
      LDP     X002  ; 急停
      ORP     M2084  ; S5異常
      ANB
      LD      M842  ; 鎖止塞起子停止
      ANI     M843  ; 鎖止塞壓緊歸
      ORB
      AND     M0  ; Auto Status
      AND     X002  ; 急停
      AND     M3  ; S5使用/不使用(ON/OFF)
      OUT     M842  ; 鎖止塞起子停止
1692  LD      M842  ; 鎖止塞起子停止
      ANI     Y007  ; S5鎖止塞起子sol
      OUT     T84 K3  ; 842
